# B&R Automation Studio project 8238
Automation Studio 4.10.2.37; technology packages: mapp 5.15.0, mappSafety 5.15.0, mappView 5.15.1, mappVision 5.15.0

## Configuration LargeLoop

CPU , AutomationRuntime E4.34, Build 4.1.2, Safety 0.0, Vc V4.33.0

### Task classes (Cpu.sw)
```
Cyclic#1 (cycle 5000 us):
  Lift_PosMo <- Robo_Drive_Control.Lift_PosMonitor.prg [disabled]
  ServerTask <- (binary)
  USB_Pmem <- (binary)
  zzClearMem <- (binary)
  can_dry1 <- (binary)
  zzSQLid <- (binary)
  Belt_Test <- (binary)
Cyclic#2 (cycle 10000 us, tolerance 10000 us):
  IO_INPUTS <- IO_INPUTS.prg
  S_COMM_IN <- S_COMM_IN.prg
  DBOUNCE <- DBOUNCE.prg
  INSERTS <- INSERTS.prg
  WEIGHT <- WEIGHT.prg
  BRING_OK <- BRING_OK.prg
  LIFTS <- LIFTS.prg
  CLOSERS <- CLOSERS.prg
  SWITCHES <- SWITCHES.prg
  OPENERS <- OPENERS.prg
  RAIL_SUB <- RAIL_SUB.prg
  ALARMS <- ALARMS.prg
  IO_OUTPUTS <- IO_OUTPUTS.prg
  S_COMM_OUT <- S_COMM_OUT.prg
  Lift_v8_1 <- Robo_Drive_Control.Lift_v8_1.prg
  custom <- custom.prg
  zzStd <- Standard.Standard.zzStd.prg
Cyclic#8 (cycle 5000 us):
  ModSlave <- ModSlave.prg
DataObjects: Param_1_5k <- Robo_Drive_Control.Param_1_5kwStar_expo.dob, assl1, arsdmsvp, arsdmhtm, arsdmsvg
Binaries: TCData, udbdef, ashwac, User, Role, OpcUaMap, asfw, arconfig, iomap, ashwd, sysconf, vcfntttf, vcfile, vcshared, vccshape, vcgclass, arial, CT1102, vcchspot, vcdsint, PCT0403, vccbtn, vcdsloc, vccovl, vccline, vcctext, vcalarm, vcbclass, vcrt, vccnum, vccstr, CT1103, arialbd, PCT0402, vcpdsw, verdanab, verdana, webserv, arsdm
Libraries: FC302, MbusTCP, sys_lib, AsARCfg, AsTCP, asstring, AsCANopen, runtime, standard, asieccon, astime, vcresman, WETCAN2, MTTypes, brsystem
```

### Hardware
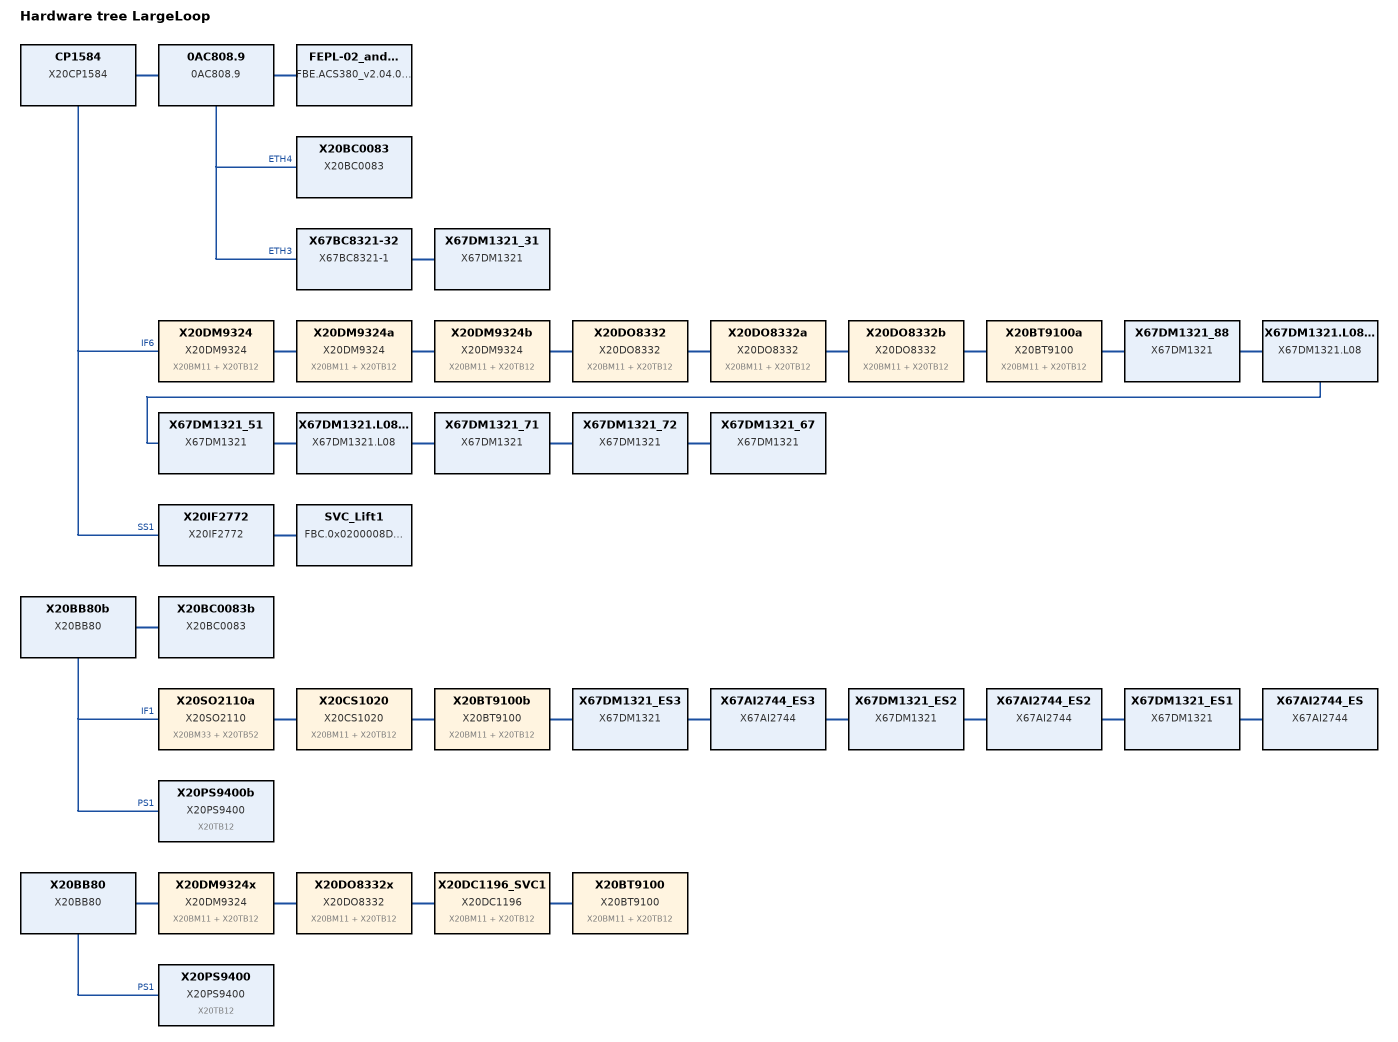
```
0AC808.9 : 0AC808.9 v1.0.0.0  [ETH1 -> CP1584.IF3 [Cable Type=PowerlinkCable, Length=10, Version=1.0.0.3]; ETH3 -> X67BC8321-32.PLK1 [Cable Type=PowerlinkCable, Length=10, Version=1.0.0.3]; ETH4 -> X20BC0083.PLK1 [Cable Type=PowerlinkCable, Length=10, Version=1.0.0.3]; ETH7 -> FEPL-02_and_ACS380_STB1.PLK1 [Cable Type=PowerlinkCable, Length=10, Version=1.0.0.3]]
CP1584 : X20CP1584 v1.9.0.0
  Connector IF2:
    ActivateDevice = 1
    Mode = Manual
    InternetAddress = 10.8.4.20
    SubnetMask = 
  Connector IF3:
    DNAConfiguration = manual
    InternetAddress = 10.0.20.20
    SubnetMask = 255.255.255.0
    ActivateIna = 1
    InaNodeNumber = 21
  Connector IF6:
    Stations = 100
  ConfigurationID = AS4_2_BaseStandard_Supertrack
  UserRamSize = 966656
  RemMemSize = 65280
  PermanentPvSize = 46956
  RemanentGlobalPvSize = 12000
  VolatileGlobalPvSize = 400000
  CyclicObjects = 200
  BRObjects = 600
  EnableUsbRemoteInstall = 1
  EnableCfRemoteInstall = 1
  Cyclic1Duration = 5000
  Cyclic2Duration = 10000
  Cyclic2Tolerance = 10000
  Cyclic8Duration = 5000
  FileDevice1
  FileDeviceName1 = USBStick
  FileDevicePath1 = /bd0\
  EthernetHostName = SupertrackPLC
  EthernetDefaultGateway = 10.8.15.254
  ActivateOpcUa = 1
  OpcUa_Security_SoftwareCertificates = 
  OpcUaInformationModels_PV_Version = 1
FEPL-02_and_ACS380_STB1 : FBE.ACS380_v2.04.0.3_FEPL-02_1.0_filerev1.0 vFFEPS10 (OrderNumber=FEPL-02 and ACS380)  [PLK1 -> 0AC808.9.ETH7 (NodeNumber=101) [Cable Type=PowerlinkCable, Length=10, Version=1.0.0.3]]
  Supervision = off
  p2201_direction = ro
  p2203_direction = ro
  p6040_direction = wo
  p6041_direction = ro
  p6042_direction = wo
  p6044_direction = ro
  p4001s07_direction = ro
  p4001s0A_direction = ro
  p401Cs48_direction = wo
  p401Cs49_direction = wo
  p4063s06_direction = wo
  p4063s09_direction = wo
  p4063s0A_direction = wo
SVC_Lift1 : FBC.0x0200008D.0x00000064.CO302A_4 v0x04.0x2A (OrderNumber=MCA105 CANopen)  [CAN1 -> X20IF2772.IF1 (NodeNumber=11)]
  p6040_connecttomaster = 6
  p6041_connecttomaster = 2
  p1400_transmissionselection = 0
  p1401_transmissionselection = 1
  p1402_transmissionselection = 0
  p1403_transmissionselection = 0
  p1800_transmissionselection = 0
  p1801_transmissionselection = 1
  p1802_transmissionselection = 0
  p1803_transmissionselection = 1
  pheartbeat_producertime = 500
  p241a_subnumber = 0x08
  p241a_parametername = 1050. Process Data Con
  p241a_objecttype = 8
  p241a_objflags = 0
  p241a_parametervalue = 
  p241asub0_parametername = 1050. Process Data Con index 0
  p241asub0_objecttype = 7
  p241asub0_accesstype = RW
  p241asub0_datatype = 6
  p241asub0_pdomapping = 0
  p241asub0_objflags = 0
  p241asub0_lowlimit = 0x0
  p241asub0_highlimit = 0x7d0
  p241asub0_parametervalue = 
  p241asub1_parametername = 1050. Process Data Con index 1
  p241asub1_objecttype = 7
  p241asub1_accesstype = RW
  p241asub1_datatype = 6
  p241asub1_pdomapping = 0
  p241asub1_objflags = 0
  p241asub1_lowlimit = 0x0
  p241asub1_highlimit = 0x7d0
  p241asub1_parametervalue = 
  p241asub2_parametername = 1050. Process Data Con index 2
  p241asub2_objecttype = 7
  p241asub2_accesstype = RW
  p241asub2_datatype = 6
  p241asub2_pdomapping = 0
  p241asub2_objflags = 0
  p241asub2_lowlimit = 0x0
  p241asub2_highlimit = 0x7d0
  p241asub2_parametervalue = 
  p241asub3_parametername = 1050. Process Data Con index 3
  p241asub3_objecttype = 7
  p241asub3_accesstype = RW
  p241asub3_datatype = 6
  p241asub3_pdomapping = 0
  p241asub3_objflags = 0
  p241asub3_lowlimit = 0x0
  p241asub3_highlimit = 0x7d0
  p241asub3_parametervalue = 
  p241asub4_parametername = 1050. Process Data Con index 4
  p241asub4_objecttype = 7
  p241asub4_accesstype = RW
  p241asub4_datatype = 6
  p241asub4_pdomapping = 0
  p241asub4_objflags = 0
  p241asub4_lowlimit = 0x0
  p241asub4_highlimit = 0x7d0
  p241asub4_parametervalue = 
  p241asub5_parametername = 1050. Process Data Con index 5
  p241asub5_objecttype = 7
  p241asub5_accesstype = RW
  p241asub5_datatype = 6
  p241asub5_pdomapping = 0
  p241asub5_objflags = 0
  p241asub5_lowlimit = 0x0
  p241asub5_highlimit = 0x7d0
  p241asub5_parametervalue = 
  p241asub6_parametername = 1050. Process Data Con index 6
  p241asub6_objecttype = 7
  p241asub6_accesstype = RW
  p241asub6_datatype = 6
  p241asub6_pdomapping = 0
  p241asub6_objflags = 0
  p241asub6_lowlimit = 0x0
  p241asub6_highlimit = 0x7d0
  p241asub6_parametervalue = 
  p241asub7_parametername = 1050. Process Data Con index 7
  p241asub7_objecttype = 7
  p241asub7_accesstype = RW
  p241asub7_datatype = 6
  p241asub7_pdomapping = 0
  p241asub7_objflags = 0
  p241asub7_lowlimit = 0x0
  p241asub7_highlimit = 0x7d0
  p241asub7_parametervalue = 
  p241b_subnumber = 0x08
  p241b_parametername = 1051. Process Data Con
  p241b_objecttype = 8
  p241b_objflags = 0
  p241b_parametervalue = 
  p241bsub0_parametername = 1051. Process Data Con index 0
  p241bsub0_objecttype = 7
  p241bsub0_accesstype = RW
  p241bsub0_datatype = 6
  p241bsub0_pdomapping = 0
  p241bsub0_objflags = 0
  p241bsub0_lowlimit = 0x0
  p241bsub0_highlimit = 0x7d0
  p241bsub0_parametervalue = 
  p241bsub1_parametername = 1051. Process Data Con index 1
  p241bsub1_objecttype = 7
  p241bsub1_accesstype = RW
  p241bsub1_datatype = 6
  p241bsub1_pdomapping = 0
  p241bsub1_objflags = 0
  p241bsub1_lowlimit = 0x0
  p241bsub1_highlimit = 0x7d0
  p241bsub1_parametervalue = 
  p241bsub2_parametername = 1051. Process Data Con index 2
  p241bsub2_objecttype = 7
  p241bsub2_accesstype = RW
  p241bsub2_datatype = 6
  p241bsub2_pdomapping = 0
  p241bsub2_objflags = 0
  p241bsub2_lowlimit = 0x0
  p241bsub2_highlimit = 0x7d0
  p241bsub2_parametervalue = 
  p241bsub3_parametername = 1051. Process Data Con index 3
  p241bsub3_objecttype = 7
  p241bsub3_accesstype = RW
  p241bsub3_datatype = 6
  p241bsub3_pdomapping = 0
  p241bsub3_objflags = 0
  p241bsub3_lowlimit = 0x0
  p241bsub3_highlimit = 0x7d0
  p241bsub3_parametervalue = 
  p241bsub4_parametername = 1051. Process Data Con index 4
  p241bsub4_objecttype = 7
  p241bsub4_accesstype = RW
  p241bsub4_datatype = 6
  p241bsub4_pdomapping = 0
  p241bsub4_objflags = 0
  p241bsub4_lowlimit = 0x0
  p241bsub4_highlimit = 0x7d0
  p241bsub4_parametervalue = 
  p241bsub5_parametername = 1051. Process Data Con index 5
  p241bsub5_objecttype = 7
  p241bsub5_accesstype = RW
  p241bsub5_datatype = 6
  p241bsub5_pdomapping = 0
  p241bsub5_objflags = 0
  p241bsub5_lowlimit = 0x0
  p241bsub5_highlimit = 0x7d0
  p241bsub5_parametervalue = 
  p241bsub6_parametername = 1051. Process Data Con index 6
  p241bsub6_objecttype = 7
  p241bsub6_accesstype = RW
  p241bsub6_datatype = 6
  p241bsub6_pdomapping = 0
  p241bsub6_objflags = 0
  p241bsub6_lowlimit = 0x0
  p241bsub6_highlimit = 0x7d0
  p241bsub6_parametervalue = 
  p241bsub7_parametername = 1051. Process Data Con index 7
  p241bsub7_objecttype = 7
  p241bsub7_accesstype = RW
  p241bsub7_datatype = 6
  p241bsub7_pdomapping = 0
  p241bsub7_objflags = 0
  p241bsub7_lowlimit = 0x0
  p241bsub7_highlimit = 0x7d0
  p241bsub7_parametervalue = 
X20BB80 : X20BB80 v1.1.0.0
X20BB80b : X20BB80 v1.1.0.0
X20BC0083 : X20BC0083 v2.14.0.0  [PLK1 -> 0AC808.9.ETH4 (NodeNumber=2) [Cable Type=PowerlinkCable, Length=10, Version=1.0.0.3]; SL -> X20BB80.SL1]
  Supervision = off
X20BC0083b : X20BC0083 v2.14.0.0  [SL -> X20BB80b.SL1]
  Supervision = off
X20BM11 : X20BM11 v1.0.0.1  [X2X1 -> CP1584.IF6]
X20BM11a : X20BM11 v1.0.0.1  [X2X1 -> X20BM11.X2X2]
X20BM11b : X20BM11 v1.0.0.1  [X2X1 -> X20BB80.IF1]
X20BM11c : X20BM11 v1.0.0.1  [X2X1 -> X20BM33b.X2X2]
X20BM11d : X20BM11 v1.0.0.1  [X2X1 -> X20BM11a.X2X2]
X20BM11e : X20BM11 v1.0.0.1  [X2X1 -> X20BM11d.X2X2]
X20BM11f : X20BM11 v1.0.0.1  [X2X1 -> X20BM11e.X2X2]
X20BM11g : X20BM11 v1.0.0.1  [X2X1 -> X20BM11b.X2X2]
X20BM11h : X20BM11 v1.0.0.1  [X2X1 -> X20BM11f.X2X2]
X20BM11i : X20BM11 v1.0.0.1  [X2X1 -> X20BM11g.X2X2]
X20BM11j : X20BM11 v1.0.0.1  [X2X1 -> X20BM11i.X2X2]
X20BM11k : X20BM11 v1.0.0.1  [X2X1 -> X20BM11h.X2X2]
X20BM11l : X20BM11 v1.0.0.1  [X2X1 -> X20BM11c.X2X2]
X20BM33b : X20BM33 v1.1.0.0  [X2X1 -> X20BB80b.IF1]
X20BT9100 : X20BT9100 v1.1.0.0  [SS1 -> X20TB12k.SS; SL -> X20BM11j.SL1]
  Supervision = off
X20BT9100a : X20BT9100 v1.1.0.0  [SS1 -> X20TB12l.SS; SL -> X20BM11k.SL1]
  Supervision = off
X20BT9100b : X20BT9100 v1.1.0.0  [SS1 -> X20TB12d.SS; SL -> X20BM11l.SL1]
  Supervision = off
X20CS1020 : X20CS1020 v1.7.0.0  [SS1 -> X20TB12o.SS; SL -> X20BM11c.SL1]
  Supervision = off
X20DC1196_SVC1 : X20DC1196 v1.3.0.0  [SS1 -> X20TB12j.SS; SL -> X20BM11i.SL1]
  FunctionModel = FunctionModel001
  Supervision = off
X20DM9324 : X20DM9324 v1.0.4.0  [SS1 -> X20TB12a.SS; SL -> X20BM11.SL1]
  Supervision = off
X20DM9324a : X20DM9324 v1.0.4.0  [SS1 -> X20TB12b.SS; SL -> X20BM11a.SL1]
  Supervision = off
X20DM9324b : X20DM9324 v1.0.4.0  [SS1 -> X20TB12e.SS; SL -> X20BM11d.SL1]
  Supervision = off
X20DM9324x : X20DM9324 v1.0.4.0  [SS1 -> X20TB12c.SS; SL -> X20BM11b.SL1]
  Supervision = off
X20DO8332 : X20DO8332 v1.0.2.0  [SS1 -> X20TB12f.SS; SL -> X20BM11e.SL1]
  Supervision = off
X20DO8332a : X20DO8332 v1.0.2.0  [SS1 -> X20TB12g.SS; SL -> X20BM11f.SL1]
  Supervision = off
X20DO8332b : X20DO8332 v1.0.2.0  [SS1 -> X20TB12i.SS; SL -> X20BM11h.SL1]
  Supervision = off
X20DO8332x : X20DO8332 v1.0.2.0  [SS1 -> X20TB12h.SS; SL -> X20BM11g.SL1]
  Supervision = off
X20IF2772 : X20IF2772 v1.5.0.0  [SS -> CP1584.SS1]
  Connector IF1:
    Baudrate = 250000
    ActivateCANIO = 0
    ActivateCanOpen = 1
    pcannodeid = 2
    pnmtstartup_bit3 = 1
    pnmtstartup_maximumbootuptime = 20
    pheartbeat_producertime = 500
    pactivatesync = 1
    pcycleperiod = 10000
    pwindowlength = 10000
    p1006_parametervalue = 0
    p1007_parametervalue = 0
    p100c_parametervalue = 1000
    p100d_parametervalue = 3
  Connector IF2:
    Baudrate = 250000
    ActivateCanOpen = 1
    pcannodeid = 3
    p1006_parametervalue = 0
    p1007_parametervalue = 0
    p100c_parametervalue = 1000
    p100d_parametervalue = 3
X20PS9400 : X20PS9400 v1.7.0.0  [SS1 -> X20TB12.SS; PS -> X20BB80.PS1]
  Supervision = off
X20PS9400b : X20PS9400 v1.7.0.0  [SS1 -> X20TB12m.SS; PS -> X20BB80b.PS1]
  Supervision = off
X20SO2110a : X20SO2110 v2.2.1.0  [SS1 -> X20TB52d.SS; SL -> X20BM33b.SL1]
  Supervision = off
  SafeModuleID = 4
X20TB12 : X20TB12 v1.0.0.0
X20TB12a : X20TB12 v1.0.0.0
X20TB12b : X20TB12 v1.0.0.0
X20TB12c : X20TB12 v1.0.0.0
X20TB12d : X20TB12 v1.0.0.0
X20TB12e : X20TB12 v1.0.0.0
X20TB12f : X20TB12 v1.0.0.0
X20TB12g : X20TB12 v1.0.0.0
X20TB12h : X20TB12 v1.0.0.0
X20TB12i : X20TB12 v1.0.0.0
X20TB12j : X20TB12 v1.0.0.0
X20TB12k : X20TB12 v1.0.0.0
X20TB12l : X20TB12 v1.0.0.0
X20TB12m : X20TB12 v1.0.0.0
X20TB12o : X20TB12 v1.0.0.0
X20TB52d : X20TB52 v1.0.0.2
X67AI2744_ES : X67AI2744 v1.3.0.0  [X2X1 -> X67DM1321_ES1.X2X2 [Cable Type=X2XCable, Length=10, Version=1.0.0.3]]
  Supervision = off
X67AI2744_ES2 : X67AI2744 v1.3.0.0  [X2X1 -> X67DM1321_ES2.X2X2 [Cable Type=X2XCable, Length=10, Version=1.0.0.3]]
  Supervision = off
X67AI2744_ES3 : X67AI2744 v1.3.0.0  [X2X1 -> X67DM1321_ES3.X2X2 [Cable Type=X2XCable, Length=10, Version=1.0.0.3]]
  Supervision = off
X67BC8321-32 : X67BC8321-1 v2.14.0.0  [PLK1 -> 0AC808.9.ETH3 (NodeNumber=1) [Cable Type=PowerlinkCable, Length=10, Version=1.0.0.3]]
  IOSupervision = off
  Direction05 = output
  Direction07 = output
  Direction08 = output
X67DM1321.L08_151 : X67DM1321.L08 v1.3.0.0  [X2X1 -> X67DM1321_88.X2X2 [Cable Type=X2XCable, Length=10, Version=1.0.0.3]]
  Supervision = off
  Direction09 = output
  Direction10 = output
  Direction11 = output
  Direction12 = output
  Direction13 = output
  Direction14 = output
  Direction15 = output
  Direction16 = output
X67DM1321.L08_152 : X67DM1321.L08 v1.3.0.0  [X2X1 -> X67DM1321_51.X2X2 [Cable Type=X2XCable, Length=10, Version=1.0.0.3]]
  Supervision = off
  Direction09 = output
  Direction10 = output
  Direction11 = output
  Direction12 = output
  Direction13 = output
  Direction14 = output
  Direction15 = output
  Direction16 = output
X67DM1321_31 : X67DM1321 v1.2.0.0  [X2X1 -> X67BC8321-32.IF1 [Cable Type=X2XCable, Length=10, Version=1.0.0.3]]
  Supervision = off
  Direction08 = output
X67DM1321_51 : X67DM1321 v1.2.0.0  [X2X1 -> X67DM1321.L08_151.X2X2 [Cable Type=X2XCable, Length=10, Version=1.0.0.3]]
  Supervision = off
  Direction05 = output
  Direction06 = output
  Direction07 = output
  Direction08 = output
X67DM1321_67 : X67DM1321 v1.2.0.0  [X2X1 -> X67DM1321_72.X2X2 [Cable Type=X2XCable, Length=10, Version=1.0.0.3]]
  Supervision = off
  Direction04 = output
  Direction05 = output
  Direction06 = output
  Direction07 = output
  Direction08 = output
X67DM1321_71 : X67DM1321 v1.2.0.0  [X2X1 -> X67DM1321.L08_152.X2X2 [Cable Type=X2XCable, Length=10, Version=1.0.0.3]]
  Supervision = off
  Direction03 = output
  Direction04 = output
  Direction05 = output
  Direction06 = output
  Direction07 = output
  Direction08 = output
X67DM1321_72 : X67DM1321 v1.2.0.0  [X2X1 -> X67DM1321_71.X2X2 [Cable Type=X2XCable, Length=10, Version=1.0.0.3]]
  Supervision = off
  Direction03 = output
  Direction04 = output
  Direction05 = output
  Direction06 = output
  Direction07 = output
  Direction08 = output
X67DM1321_88 : X67DM1321 v1.2.0.0  [X2X1 -> X20BT9100a.X2X1 [Cable Type=X2XCable, Length=10, Version=1.0.0.3]]
  Supervision = off
  Direction06 = output
  Direction07 = output
  Direction08 = output
X67DM1321_ES1 : X67DM1321 v1.2.0.0  [X2X1 -> X67AI2744_ES2.X2X2 [Cable Type=X2XCable, Length=10, Version=1.0.0.3]]
  Supervision = off
  Direction01 = output
  Direction02 = output
  Direction05 = output
  Direction06 = output
  Direction07 = output
  Direction08 = output
X67DM1321_ES2 : X67DM1321 v1.2.0.0  [X2X1 -> X67AI2744_ES3.X2X2 [Cable Type=X2XCable, Length=10, Version=1.0.0.3]]
  Supervision = off
  Direction01 = output
  Direction02 = output
  Direction05 = output
  Direction06 = output
  Direction07 = output
  Direction08 = output
X67DM1321_ES3 : X67DM1321 v1.2.0.0  [X2X1 -> X20BT9100b.X2X1 [Cable Type=X2XCable, Length=10, Version=1.0.0.3]]
  Supervision = off
  Direction01 = output
  Direction02 = output
  Direction05 = output
  Direction06 = output
  Direction07 = output
  Direction08 = output
```

### IoMap.iom - CP1584/IoMap.iom
```iecst
(********************************************************************
 * COPYRIGHT --
 ********************************************************************
 * File: IoMap.iom
 * Author: Dave
 * Created: November 19, 2010
 ********************************************************************
 * IO mapping file
 ********************************************************************)
VAR_CONFIG
	OK[1] AT %IX."X20DM9324x".ModuleOk;
	OK[3] AT %IX."X20DO8332x".ModuleOk;
	X[1].X01 AT %IX."X20DM9324x".DigitalInput01; (*Emergency stops Ok*)
	X[1].X02 AT %IX."X20DM9324x".DigitalInput02; (*Motor overloads*)
	X[1].X03 AT %IX."X20DM9324x".DigitalInput03; (*SR1 Ok*)
	X[1].X04 AT %IX."X20DM9324x".DigitalInput04; (*Spare*)
	X[1].X05 AT %IX."X20DM9324x".DigitalInput05; (*STB1 - PX*)
	X[1].X06 AT %IX."X20DM9324x".DigitalInput06; (*STB2 -PX*)
	X[1].X07 AT %IX."X20DM9324x".DigitalInput07; (*ES2 - Emergency stop*)
	X[1].X08 AT %IX."X20DM9324x".DigitalInput08; (*ES3 - Emergency stop*)
	Y[1].Y01 AT %QX."X20DM9324x".DigitalOutput01; (*Alarm beacon*)
	Y[1].Y02 AT %QX."X20DM9324x".DigitalOutput02; (*Spare*)
	Y[1].Y03 AT %QX."X20DM9324x".DigitalOutput03; (*Spare*)
	Y[1].Y04 AT %QX."X20DM9324x".DigitalOutput04; (*Spare*)
	Y[3].Y01 AT %QX."X20DO8332x".DigitalOutput01; (*STB1 - Run*)
	Y[3].Y02 AT %QX."X20DO8332x".DigitalOutput02; (*STB2 - Run*)
	Y[3].Y03 AT %QX."X20DO8332x".DigitalOutput03; (*Spare*)
	Y[3].Y04 AT %QX."X20DO8332x".DigitalOutput04; (*Spare*)
	Y[3].Y05 AT %QX."X20DO8332x".DigitalOutput05; (*Spare*)
	Y[3].Y06 AT %QX."X20DO8332x".DigitalOutput06; (*SVC1 - Carriage stop*)
	Y[3].Y07 AT %QX."X20DO8332x".DigitalOutput07; (*Spare*)
	Y[3].Y08 AT %QX."X20DO8332x".DigitalOutput08; (*Spare*)
	X[32].X01 AT %IX."X67BC8321-32".IF1.ST1.DigitalInput01; (*SVC1 - Over travel top*)
	X[32].X02 AT %IX."X67BC8321-32".IF1.ST1.DigitalInput02; (*Spare*)
	X[32].X03 AT %IX."X67BC8321-32".IF1.ST1.DigitalInput03; (*SVC1 - Over travel bottom*)
	Cyclic#1.X[32].X04 AT %IX."X67BC8321-32".IF1.ST1.DigitalInput04; (*SVC1 - Reference switch*)
	Y[32].Y05 AT %QX."X67BC8321-32".IF1.ST1.DigitalOutput05; (*SVC1 - Rail end stop (Empty bag in)*)
	Y[32].Y07 AT %QX."X67BC8321-32".IF1.ST1.DigitalOutput07; (*Spare*)
	Y[32].Y08 AT %QX."X67BC8321-32".IF1.ST1.DigitalOutput08; (*SVC1 - Open buffer stop*)
	OK[31] AT %IX."X67DM1321_31".ModuleOk;
	X[31].X01 AT %IX."X67DM1321_31".DigitalInput01; (*Spare*)
	X[31].X02 AT %IX."X67DM1321_31".DigitalInput02; (*Spare*)
	X[31].X03 AT %IX."X67DM1321_31".DigitalInput03; (*Spare*)
	X[31].X04 AT %IX."X67DM1321_31".DigitalInput04; (*SVC1 Bag arrive on carriage*)
	X[31].X05 AT %IX."X67DM1321_31".DigitalInput05; (*SVC1 Bag on carriage*)
	X[31].X06 AT %IX."X67DM1321_31".DigitalInput06; (*SVC1 Rail align receive*)
	X[31].X07 AT %IX."X67DM1321_31".DigitalInput07; (*SVC1 Rail align release*)
	Y[31].Y08 AT %QX."X67DM1321_31".DigitalOutput08; (*Spare*)
	X[32].X06 AT %IX."X67BC8321-32".IF1.ST1.DigitalInput06; (*SVC1 - Bag at buffer*)
	X[88].X01 AT %IX."X67DM1321_88".DigitalInput01; (*Spare*)
	X[88].X02 AT %IX."X67DM1321_88".DigitalInput02; (*STRF1 - Bag at buffer*)
	X[88].X03 AT %IX."X67DM1321_88".DigitalInput03; (*STRF1 - Bag arrive*)
	X[88].X04 AT %IX."X67DM1321_88".DigitalInput04; (*STRF1 - Bag past point*)
	Y[88].Y06 AT %QX."X67DM1321_88".DigitalOutput06; (*STRF1 - Open buffer*)
	Y[88].Y07 AT %QX."X67DM1321_88".DigitalOutput07; (*STRF1 - Select line B*)
	Y[88].Y08 AT %QX."X67DM1321_88".DigitalOutput08; (*STRF1 - Select line A*)
	OK[88] AT %IX."X67DM1321_88".ModuleOk;
	X[151].X01 AT %IX."X67DM1321.L08_151".DigitalInput01; (*SDC1 - Bag at buffer*)
	X[151].X02 AT %IX."X67DM1321.L08_151".DigitalInput02; (*SDC1 - Bag at Discharger*)
	X[151].X03 AT %IX."X67DM1321.L08_151".DigitalInput03; (*SDC1 - Bag released*)
	X[151].X04 AT %IX."X67DM1321.L08_151".DigitalInput04; (*SDC1 - Bag empty*)
	X[151].X05 AT %IX."X67DM1321.L08_151".DigitalInput05; (*Spare*)
	X[151].X06 AT %IX."X67DM1321.L08_151".DigitalInput06; (*SDC1 - Drop load pushbutton*)
	X[151].X07 AT %IX."X67DM1321.L08_151".DigitalInput07; (*Spare*)
	X[151].X08 AT %IX."X67DM1321.L08_151".DigitalInput08; (*Spare*)
	Y[151].Y01 AT %QX."X67DM1321.L08_151".DigitalOutput09; (*SDC1 - Open buffer stop*)
	Y[151].Y02 AT %QX."X67DM1321.L08_151".DigitalOutput10; (*SDC1 - Bag steady*)
	Y[151].Y03 AT %QX."X67DM1321.L08_151".DigitalOutput11; (*SDC1 - Open bag*)
	Y[151].Y04 AT %QX."X67DM1321.L08_151".DigitalOutput12; (*SDC1 - Open stop*)
	Y[151].Y05 AT %QX."X67DM1321.L08_151".DigitalOutput13; (*SDC1 - Bag closer*)
	Y[151].Y06 AT %QX."X67DM1321.L08_151".DigitalOutput14; (*SSB1 Bag catch*)
	Y[151].Y07 AT %QX."X67DM1321.L08_151".DigitalOutput15; (*SSB1 Close bag*)
	Y[151].Y08 AT %QX."X67DM1321.L08_151".DigitalOutput16; (*SDC1 - Pushbutton lamp*)
	OK[151] AT %IX."X67DM1321.L08_151".ModuleOk;
	X[88].X05 AT %IX."X67DM1321_88".DigitalInput05; (*STRF1 - Bag released*)
	X[51].X01 AT %IX."X67DM1321_51".DigitalInput01; (*SPN1 - Bag arrive line 1*)
	X[51].X02 AT %IX."X67DM1321_51".DigitalInput02; (*SPN1 - Bag arrive line 2*)
	X[51].X03 AT %IX."X67DM1321_51".DigitalInput03; (*SPN1 - Bag arrive line 3*)
	X[51].X04 AT %IX."X67DM1321_51".DigitalInput04; (*Spare*)
	Y[51].Y05 AT %QX."X67DM1321_51".DigitalOutput05; (*SPN1 - Select line 3*)
	Y[51].Y06 AT %QX."X67DM1321_51".DigitalOutput06; (*SPN1 - Select line 2*)
	Y[51].Y07 AT %QX."X67DM1321_51".DigitalOutput07; (*SPN1 - Reset line 3*)
	Y[51].Y08 AT %QX."X67DM1321_51".DigitalOutput08; (*SPN1 - Reset line 2*)
	OK[51] AT %IX."X67DM1321_51".ModuleOk;
	X[152].X01 AT %IX."X67DM1321.L08_152".DigitalInput01; (*SDC2 - Bag at buffer*)
	X[152].X02 AT %IX."X67DM1321.L08_152".DigitalInput02; (*SDC2 - Bag at Discharger*)
	X[152].X03 AT %IX."X67DM1321.L08_152".DigitalInput03; (*SDC2 - Bag released*)
	X[152].X04 AT %IX."X67DM1321.L08_152".DigitalInput04; (*SDC2 - Bag empty*)
	X[152].X05 AT %IX."X67DM1321.L08_152".DigitalInput05; (*Spare*)
	X[152].X06 AT %IX."X67DM1321.L08_152".DigitalInput06; (*SDC2 - Drop load pushbutton*)
	X[152].X07 AT %IX."X67DM1321.L08_152".DigitalInput07; (*Spare*)
	X[152].X08 AT %IX."X67DM1321.L08_152".DigitalInput08; (*Spare*)
	Y[152].Y01 AT %QX."X67DM1321.L08_152".DigitalOutput09; (*SDC2 - Open buffer stop*)
	Y[152].Y02 AT %QX."X67DM1321.L08_152".DigitalOutput10; (*SDC2 - Bag steady*)
	Y[152].Y03 AT %QX."X67DM1321.L08_152".DigitalOutput11; (*SDC2 - Open bag*)
	Y[152].Y04 AT %QX."X67DM1321.L08_152".DigitalOutput12; (*SDC2 - Open stop*)
	Y[152].Y05 AT %QX."X67DM1321.L08_152".DigitalOutput13; (*SDC2 - Bag closer*)
	Y[152].Y06 AT %QX."X67DM1321.L08_152".DigitalOutput14; (*SSB2 Bag catch*)
	Y[152].Y07 AT %QX."X67DM1321.L08_152".DigitalOutput15; (*SSB2 Close bag*)
	Y[152].Y08 AT %QX."X67DM1321.L08_152".DigitalOutput16; (*SDC2 - Pushbutton lamp*)
	OK[152] AT %IX."X67DM1321.L08_152".ModuleOk;
	X[71].X01 AT %IX."X67DM1321_71".DigitalInput01; (*SPF1 - Bag at line 1*)
	X[71].X02 AT %IX."X67DM1321_71".DigitalInput02; (*SPF1 - Bag at line 2*)
	Y[71].Y03 AT %QX."X67DM1321_71".DigitalOutput03; (*SPF1 - Open stop  line 1*)
	Y[71].Y04 AT %QX."X67DM1321_71".DigitalOutput04; (*SPF1 - Open stop  line 2*)
	Y[71].Y05 AT %QX."X67DM1321_71".DigitalOutput05; (*Spare*)
	Y[71].Y06 AT %QX."X67DM1321_71".DigitalOutput06; (*SPF1 - Select line 2*)
	Y[71].Y07 AT %QX."X67DM1321_71".DigitalOutput07; (*Spare*)
	Y[71].Y08 AT %QX."X67DM1321_71".DigitalOutput08; (*SPF1 - Reset line 2*)
	OK[71] AT %IX."X67DM1321_71".ModuleOk; (*Module status (3 = module present)*)
	X[72].X01 AT %IX."X67DM1321_72".DigitalInput01; (*SPF1 - Bag at line 3*)
	X[72].X02 AT %IX."X67DM1321_72".DigitalInput02; (*SPF1 - Bag released*)
	Y[72].Y03 AT %QX."X67DM1321_72".DigitalOutput03; (*SPF1 - Open stop  line 3*)
	Y[72].Y04 AT %QX."X67DM1321_72".DigitalOutput04; (*Spare*)
	Y[72].Y05 AT %QX."X67DM1321_72".DigitalOutput05; (*SPF1 - Select line 3*)
	Y[72].Y06 AT %QX."X67DM1321_72".DigitalOutput06; (*Spare*)
	Y[72].Y07 AT %QX."X67DM1321_72".DigitalOutput07; (*SPF1 - Reset line 3*)
	Y[72].Y08 AT %QX."X67DM1321_72".DigitalOutput08; (*Spare*)
	OK[72] AT %IX."X67DM1321_72".ModuleOk; (*Module status (3 = module present)*)
	X[67].X01 AT %IX."X67DM1321_67".DigitalInput01; (*SVC2 - Bag at buffer line B*)
	X[67].X02 AT %IX."X67DM1321_67".DigitalInput02; (*SVC2 - Bag at buffer line A*)
	X[67].X03 AT %IX."X67DM1321_67".DigitalInput03; (*STRN1 - Bag past point*)
	Y[67].Y05 AT %QX."X67DM1321_67".DigitalOutput05; (*SVC2 - Open buffer line B*)
	Y[67].Y06 AT %QX."X67DM1321_67".DigitalOutput06; (*SVC2 - Open buffer line A*)
	Y[67].Y07 AT %QX."X67DM1321_67".DigitalOutput07; (*STRN1 - Select line B*)
	Y[67].Y08 AT %QX."X67DM1321_67".DigitalOutput08; (*STRN1 - Select line A*)
	OK[67] AT %IX."X67DM1321_67".ModuleOk;
	Y[67].Y04 AT %QX."X67DM1321_67".DigitalOutput04; (*SVC2 - Safety stops*)
	X[303].X03 AT %IX."X67DM1321_ES3".DigitalInput03; (*ES3 - Pushbutton*)
	X[303].X04 AT %IX."X67DM1321_ES3".DigitalInput04; (*Spare*)
	Y[303].Y01 AT %QX."X67DM1321_ES3".DigitalOutput01; (*ES3 - Lamp*)
	Y[303].Y02 AT %QX."X67DM1321_ES3".DigitalOutput02; (*ES3 - Open door*)
	Y[303].Y05 AT %QX."X67DM1321_ES3".DigitalOutput05; (*Spare*)
	Y[303].Y06 AT %QX."X67DM1321_ES3".DigitalOutput06; (*Spare*)
	Y[303].Y07 AT %QX."X67DM1321_ES3".DigitalOutput07; (*Spare*)
	Y[303].Y08 AT %QX."X67DM1321_ES3".DigitalOutput08; (*Spare*)
	OK[303] AT %IX."X67DM1321_ES3".ModuleOk;
	X[302].X03 AT %IX."X67DM1321_ES2".DigitalInput03; (*ES2 - Pushbutton*)
	X[302].X04 AT %IX."X67DM1321_ES2".DigitalInput04; (*Spare*)
	Y[302].Y01 AT %QX."X67DM1321_ES2".DigitalOutput01; (*ES2 - Lamp*)
	Y[302].Y02 AT %QX."X67DM1321_ES2".DigitalOutput02; (*ES2 - Open door*)
	Y[302].Y05 AT %QX."X67DM1321_ES2".DigitalOutput05; (*Spare*)
	Y[302].Y06 AT %QX."X67DM1321_ES2".DigitalOutput06; (*Spare*)
	Y[302].Y07 AT %QX."X67DM1321_ES2".DigitalOutput07; (*Spare*)
	Y[302].Y08 AT %QX."X67DM1321_ES2".DigitalOutput08; (*Spare*)
	OK[302] AT %IX."X67DM1321_ES2".ModuleOk;
	X[301].X03 AT %IX."X67DM1321_ES1".DigitalInput03; (*ES1 - Pushbutton*)
	X[301].X04 AT %IX."X67DM1321_ES1".DigitalInput04; (*Spare*)
	Y[301].Y01 AT %QX."X67DM1321_ES1".DigitalOutput01; (*ES1 - Lamp*)
	Y[301].Y02 AT %QX."X67DM1321_ES1".DigitalOutput02; (*ES1 - Open door*)
	Y[301].Y05 AT %QX."X67DM1321_ES1".DigitalOutput05; (*Spare*)
	Y[301].Y06 AT %QX."X67DM1321_ES1".DigitalOutput06; (*Spare*)
	Y[301].Y07 AT %QX."X67DM1321_ES1".DigitalOutput07; (*Spare*)
	Y[301].Y08 AT %QX."X67DM1321_ES1".DigitalOutput08; (*Spare*)
	OK[301] AT %IX."X67DM1321_ES1".ModuleOk;
	RB[1].Lift.CAN.ModuleOk AT %IX."SVC_Lift1".ModuleOk;
	RB[1].Lift.CAN.NodeStatus AT %IW."SVC_Lift1".NodeStatus;
	RB[1].Lift.CAN.ControlWord AT %QW."SVC_Lift1".CTW_6040_Out;
	RB[1].Lift.CAN.StatusWord AT %IW."SVC_Lift1".STW_6041;
	RB[1].Lift.CAN.TargetVelocity AT %QW."SVC_Lift1".TargetVelocity_6042_Out;
	RB[1].Lift.CAN.ControlEffort AT %IW."SVC_Lift1".ControlEffort_MAV_6044;
	RB[1].Lift.ModuleOK AT %IX."X20DC1196_SVC1".ModuleOk;
	RB[1].Lift.Encoder AT %ID."X20DC1196_SVC1".Encoder01;
  Cyclic#1.ABB_EPL[1].Comm.ModuleOk AT %IX."FEPL-02_and_ACS380_STB1".ModuleOk;
	Cyclic#1.ABB_EPL[1].Parameters.Write.Motor_NominalCurrent_9906 AT %QD."FEPL-02_and_ACS380_STB1"._9906_Motor_nominal_current_I4063_S06Out;
	Cyclic#1.ABB_EPL[1].Parameters.Write.Motor_NominalPower_9910 AT %QD."FEPL-02_and_ACS380_STB1"._9910_Motor_nominal_power_I4063_S0AOut;
	Cyclic#1.ABB_EPL[1].Parameters.Write.Motor_NominalSpeed_9909 AT %QD."FEPL-02_and_ACS380_STB1"._9909_Motor_nominal_speed_I4063_S09Out;
	Cyclic#1.ABB_EPL[1].Comm.ControlWord AT %QW."FEPL-02_and_ACS380_STB1".ControlWord_I6040Out;
	Cyclic#1.ABB_EPL[1].Comm.StatusWord AT %IW."FEPL-02_and_ACS380_STB1".StatusWord_I6041;
	Cyclic#1.ABB_EPL[1].Comm.ActVelocity AT %IW."FEPL-02_and_ACS380_STB1".VlVelocityActualValue_I6044;
	Cyclic#1.ABB_EPL[1].Comm.ActCurrent AT %ID."FEPL-02_and_ACS380_STB1"._0107_Motor_current_I4001_S07;
	Cyclic#1.ABB_EPL[1].Comm.ActTorque AT %ID."FEPL-02_and_ACS380_STB1"._0110_Motor_torque_I4001_S0A;
	Cyclic#1.ABB_EPL[1].Comm.ErrorCode AT %IW."FEPL-02_and_ACS380_STB1".VendorSpecificAlarmCodes_I2203;
	Cyclic#1.ABB_EPL[1].Parameters.Write.Ramp_AccTime1_2872 AT %QD."FEPL-02_and_ACS380_STB1"._2872_Freq_acceleration_time_1_I401C_S48Out;
	Cyclic#1.ABB_EPL[1].Parameters.Write.Ramp_DecTime1_2873 AT %QD."FEPL-02_and_ACS380_STB1"._2873_Freq_deceleration_time_1_I401C_S49Out;
	Cyclic#1.ABB_EPL[1].Comm.TargetVelocity AT %QW."FEPL-02_and_ACS380_STB1".VlTargetVelocity_I6042Out;
END_VAR
```

- Safety project (password-protected, skipped)

## Configuration eVue

CPU 5APC2200.AL14-000, AutomationRuntime D4.91, Build 4.1.2, Safety 0.0, Vc V4.62.0

### Task classes (Cpu.sw)
```
Cyclic#1 (cycle 1000 us, tolerance 2000 us):
  moduleWatc <- Standard.ModuleLogger.moduleWatch.prg
  USB_Pmem <- (binary)
  zzClearMem <- (binary)
  can_dry1 <- (binary)
  zzSQLid <- (binary)
  IO_Info <- (binary)
  IOLink_Dri <- (binary)
  SCANNERS <- (binary)
  SafetyUI <- (binary)
Cyclic#2 (cycle 12000 us, tolerance 12000 us):
  S_COMM_IN <- S_COMM_IN.prg
  IO_INPUTS <- IO_INPUTS.prg
  DBOUNCE <- DBOUNCE.prg
  custom <- custom.prg
  BELT_TO_TR <- BELT_TO_TRANSFER.prg
  CONVEYOR_M <- CONVEYOR_MAP.prg
  SAFETY_ZON <- SAFETY_ZONES.prg
  RAIL_SUB <- RAIL_SUB.prg
  LOADCELLS <- LOADCELLS.prg
  INSERTS <- INSERTS.prg
  WEIGHT <- WEIGHT.prg
  CLOSERS <- CLOSERS.prg
  OPENERS <- OPENERS.prg
  SWITCHES <- SWITCHES.prg
  LIFTS <- LIFTS.prg
  BRING_OK <- BRING_OK.prg
  Permenant <- Standard.Settings.Permenant.prg
  Lift_v8_1 <- Robo_Drive_Control.Lift_v8_1.prg [disabled]
  zzStd1 <- Standard.Standard.zzStd.prg
  FuseManage <- Standard.IOLink.Fuses.FuseManagement.prg
  Camera_Dri <- Standard.Barcode_BnR.Camera_Driver.prg [disabled]
  HoistServe <- Standard.HoistLibrary.HoistServer.prg
  hlKanLink <- Standard.Kanlink.KGFramework.Pkg_hlKanLink.hlKanLink.prg
Cyclic#4 (cycle 12000 us, tolerance 12000 us):
  WARNINGS <- WARNINGS.prg
Cyclic#5 (cycle 12000 us, tolerance 12000 us):
  ALARMS <- ALARMS.prg
Cyclic#6 (cycle 54000 us, tolerance 54000 us):
  zz_Kanlink <- Standard.Kanlink.zz_KanlinkConfig.prg
  Kan_Driver <- Standard.Kanlink.Kan_Driver.prg
  mnEth <- Standard.Kanlink.KGFramework.Pkg_mnEth.mnEth.prg
  svCPCache <- Standard.Kanlink.KGFramework.Pkg_svCPCache.svCPCache.prg
  kanlink_ma <- Standard.Kanlink.kanlink_map.prg
Cyclic#7 (cycle 102000 us, tolerance 102000 us):
  Contactron <- Standard.IOLink.Contactron.Contactron.prg
  httpServer <- http_Lib.httpServer.prg
Cyclic#8 (cycle 12000 us, tolerance 30000000 us):
  IO_OUTPUTS <- IO_OUTPUTS.prg
  S_COMM_OUT <- S_COMM_OUT.prg
  ModSlave <- COMMUNICATION.ModSlave.prg
  udpComm <- COMMUNICATION.UdpComm.prg
  tcpComm <- COMMUNICATION.TcpComm.prg
  udpComm_di <- SortingSpecial.udpComm_disp.prg
  zzGetTime <- CSP_Control.zzGetTime.prg
  OPCuAClien <- OPCuA_Client.OPCuAClient.prg
  mappSafety <- Safety.mappSafety.prg
  AccessCont <- Safety.AccessControl.prg
  Safety <- Safety.Safety.prg
  ABB_Driver <- Standard.ABB_EPL.ABB_Driver.prg
DataObjects: Param_1_5k <- Robo_Drive_Control.Param_1_5kwStar.dob [disabled], assl1, arsdmsvp, arsdmhtm, arsdmsvg
Binaries: mvLoader, TCLang, arflatprv, arcoal, TCData, udbdef, arsvcreg, FWRules, OpcUaSrv, Config, TC, viComp, Settings, viAppBCDE, cUnits, User, Role, sysconf, ashwd, arconfig, asfw, ashwac, iomap, Settings_1, Config_1, asiol1, asiol3, asiol2, asiol20, asiol17, asiol4, asiol19, asiol24, asiol30, asiol9, asiol12, asiol5, asiol29, asiol18, asiol16, asiol22, asiol6, asiol11, asiol28, asiol8, asiol26, asiol7, asiol15, asiol21, asiol10, asiol13, asiol32, asiol25, asiol31, asiol14, asiol23, asiol27, OpcUaMap, vcfntttf, vcfile, vcshared, vccshape, vcgclass, arial, CT1102, vcchspot, vcdsint, PCT0403, vccbtn, vcdsloc, vccovl, vccline, vcctext, vcalarm, vcbclass, vcrt, vccnum, vccstr, CT1103, arialbd, PCT0402, vcpdsw, verdanab, verdana, webserv, arsdm
Libraries: AsOpcUac, OPCuAClnt, FC302, standard, runtime, OPERATOR, AsTime, AsString, sys_lib, AsTCP, AsARCfg, AsIecCon, AsBrStr, FileIO, AsBrMath, CAN_Lib, AsUDP, MTTypes, brsystem, MpAudit, MpBase, DataObj, AsXml, MTBasics, MpServer, ArSsl, ArUser, ViBase, AsZip, powerlnk, AsEPL, AsETH, AsIODiag, AsHttp, AsIOAcc, AsIoTrc, FileMgr, AsIOLink, AsCANopen, AsIO, MbusTCP, SfDomain, KGstdLib, KGlibMsg, mnParamLib, KanLinkLib, KL_UserLib, libTestUse, AsBrWStr, ETHERNET, AsArLog, AsUSB, AsMem, AsDb, KanHttp, AsFifo, eVueLib, SfDomDrv, MpSfDomMgr, SfDomVis, SupFile, vcresman, WETCAN2, AsIOMMan, IOLinkLib, ABB_EPL
```

### Hardware
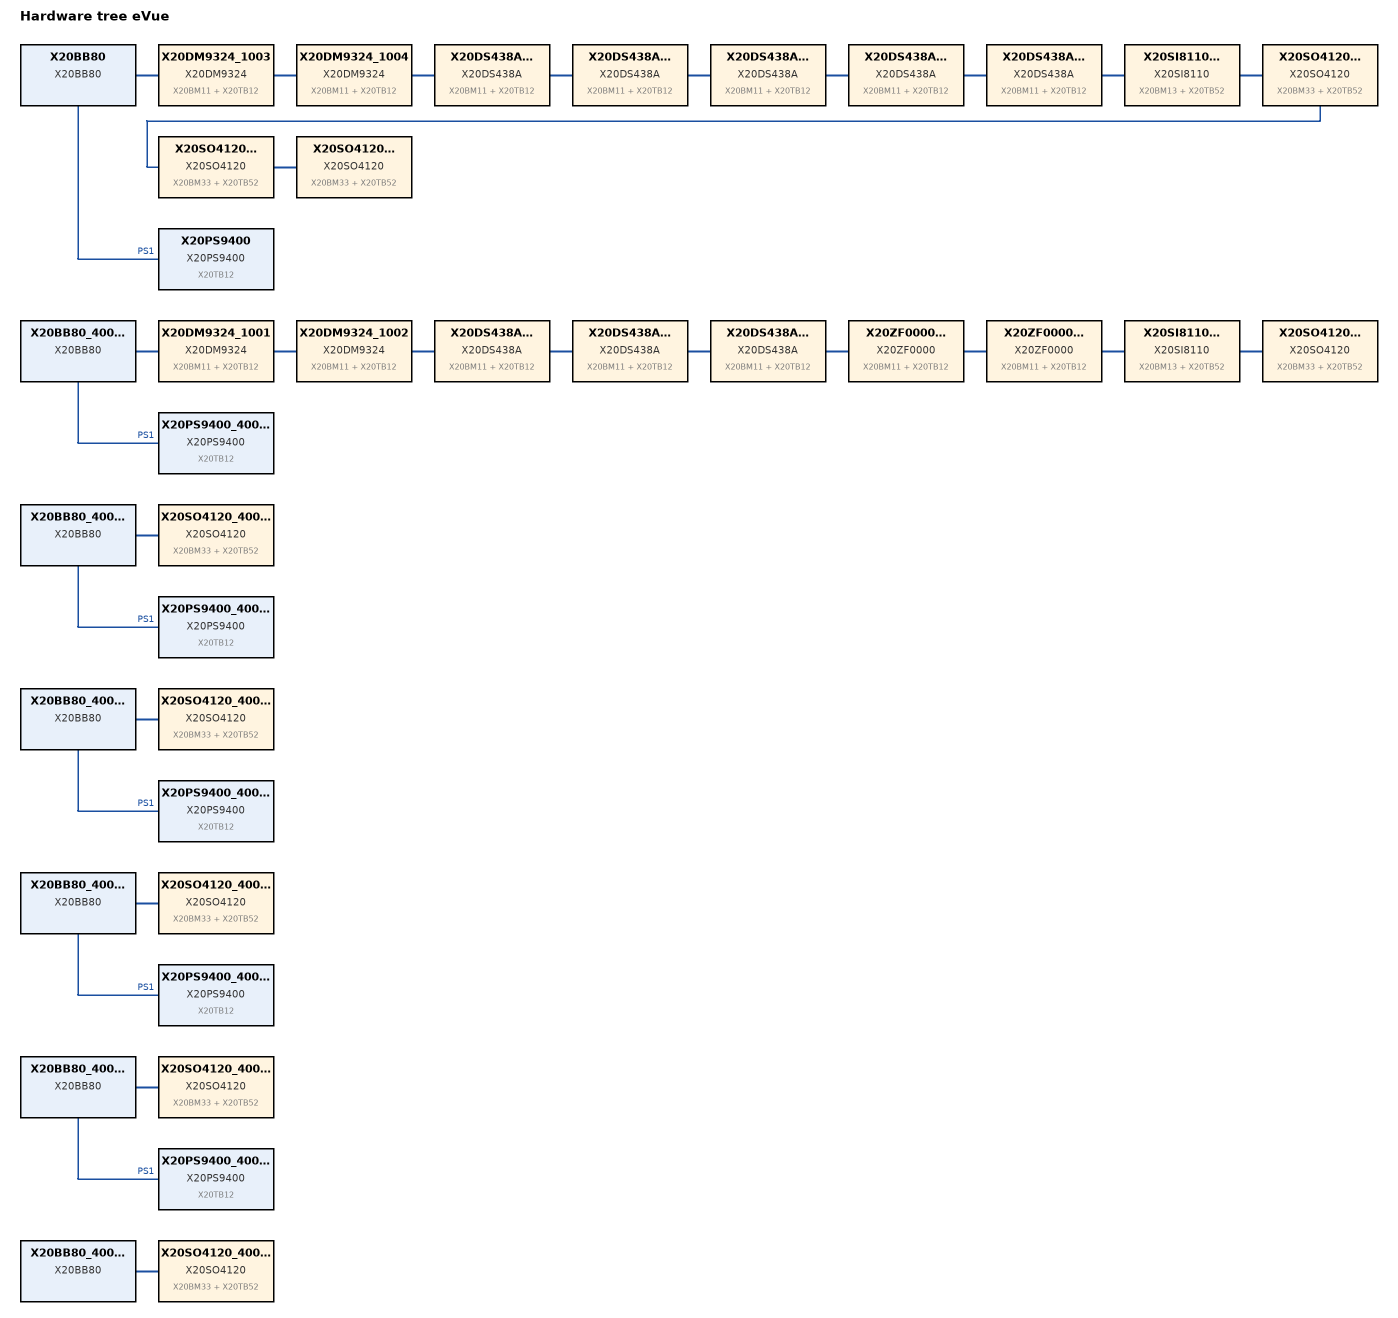
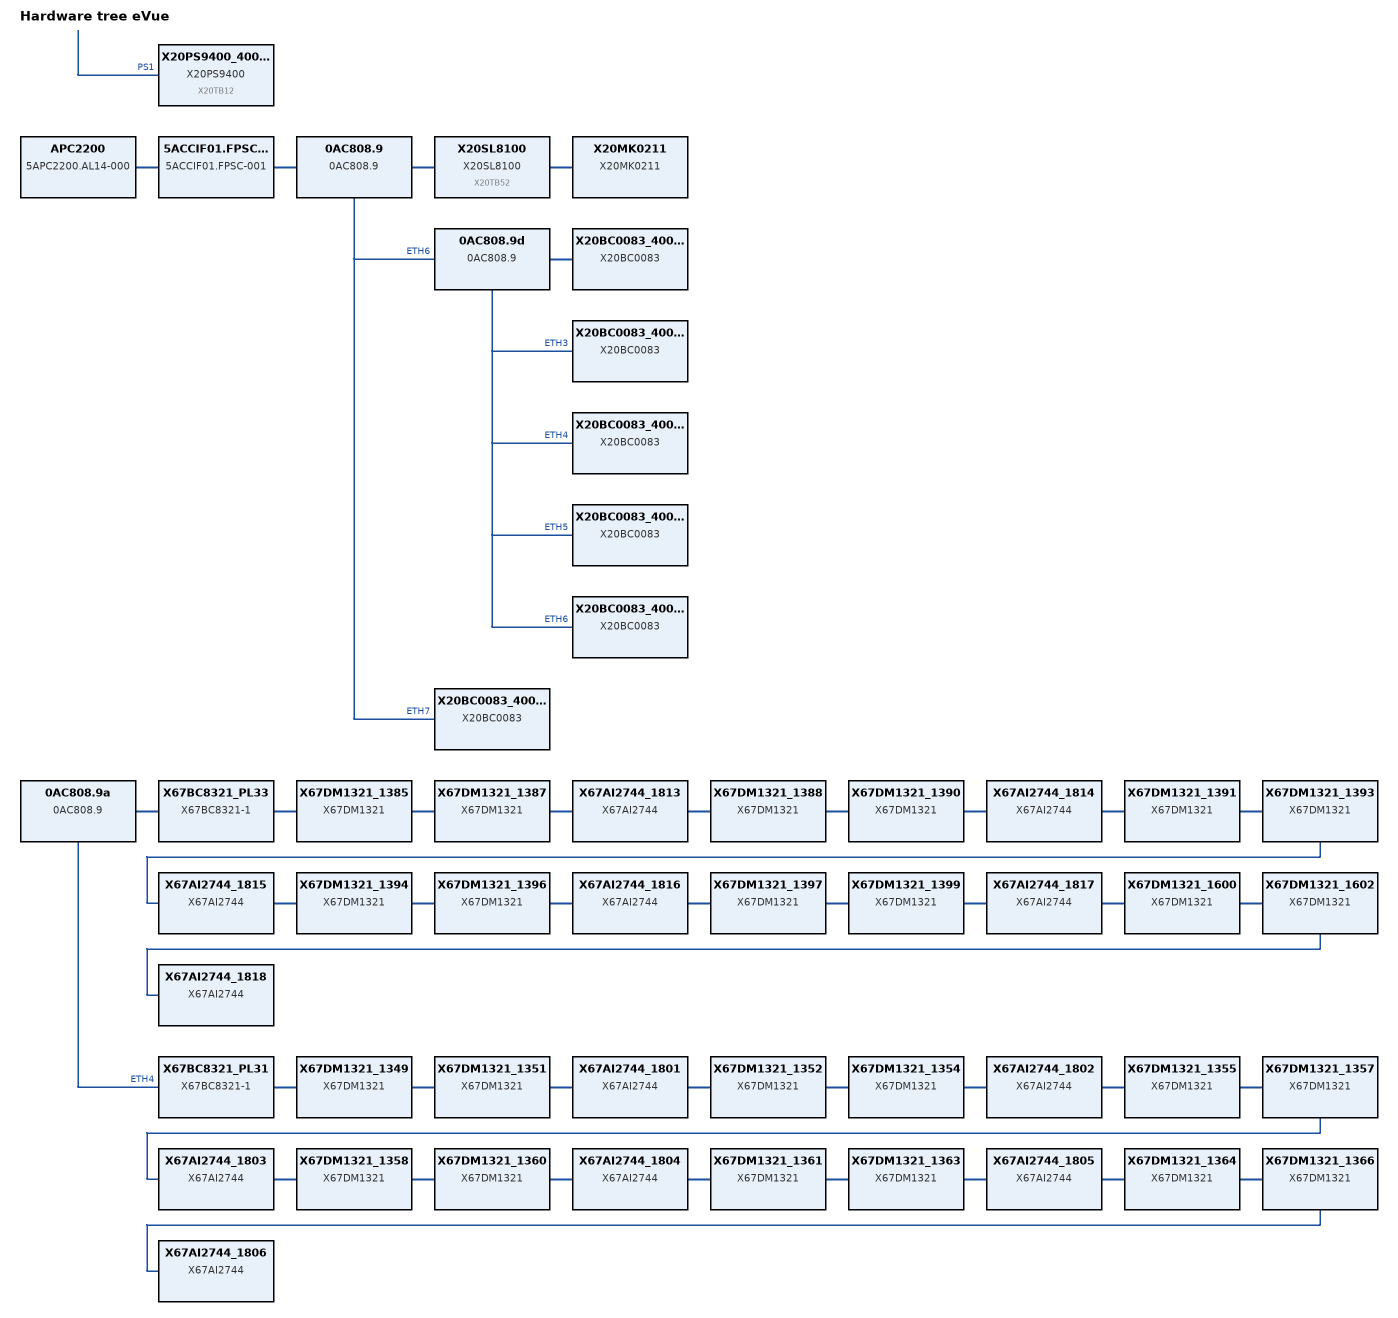
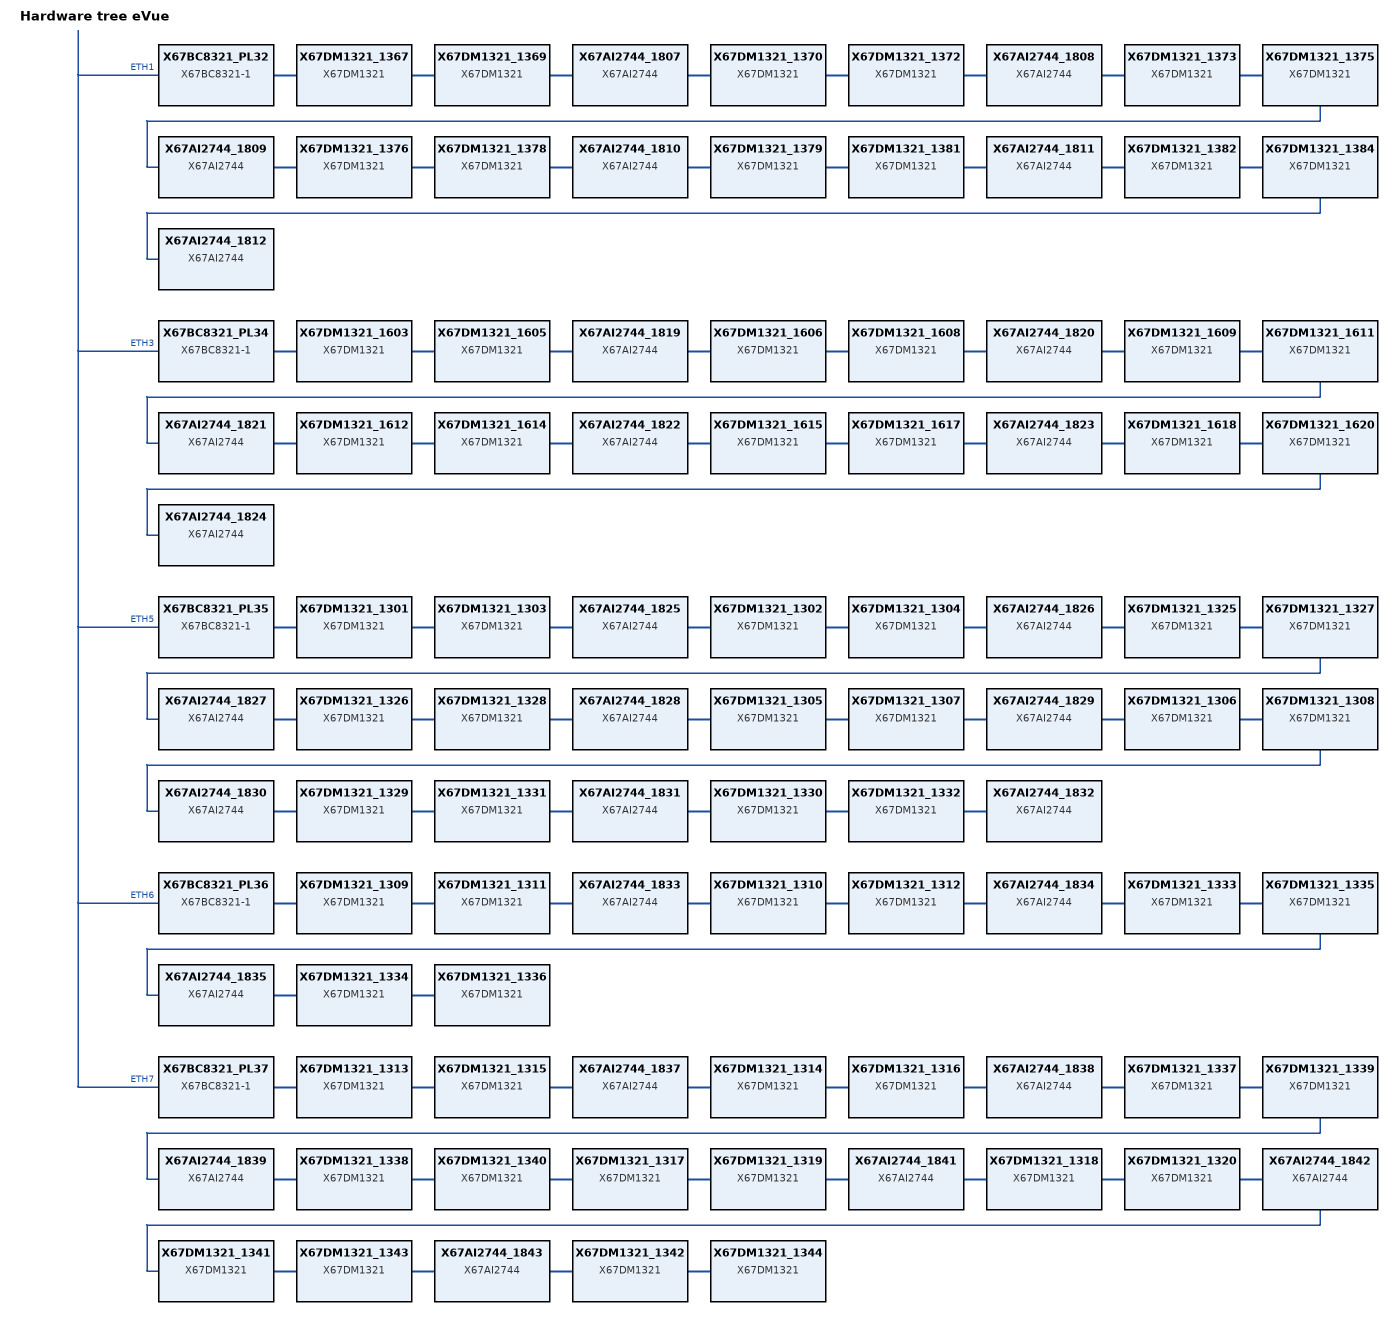
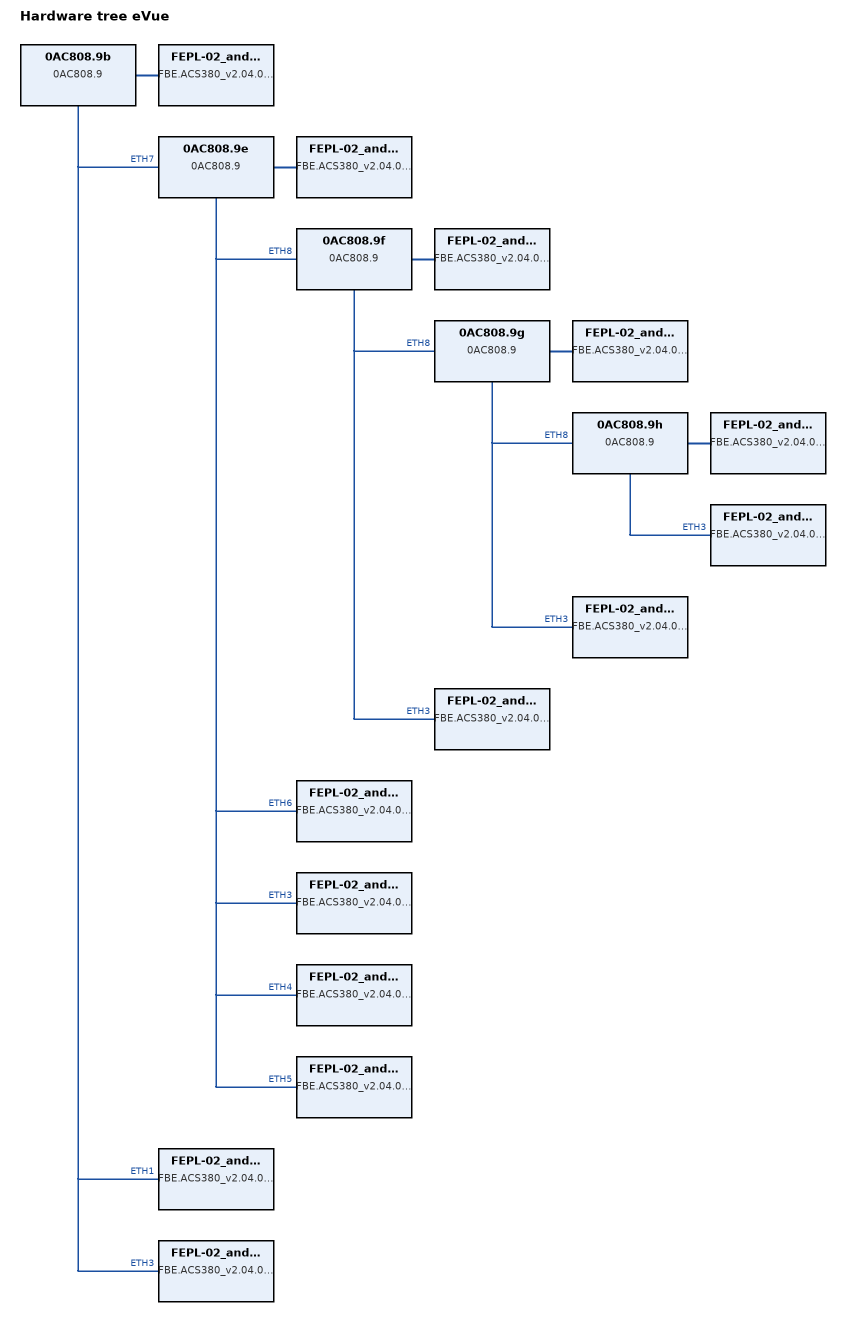
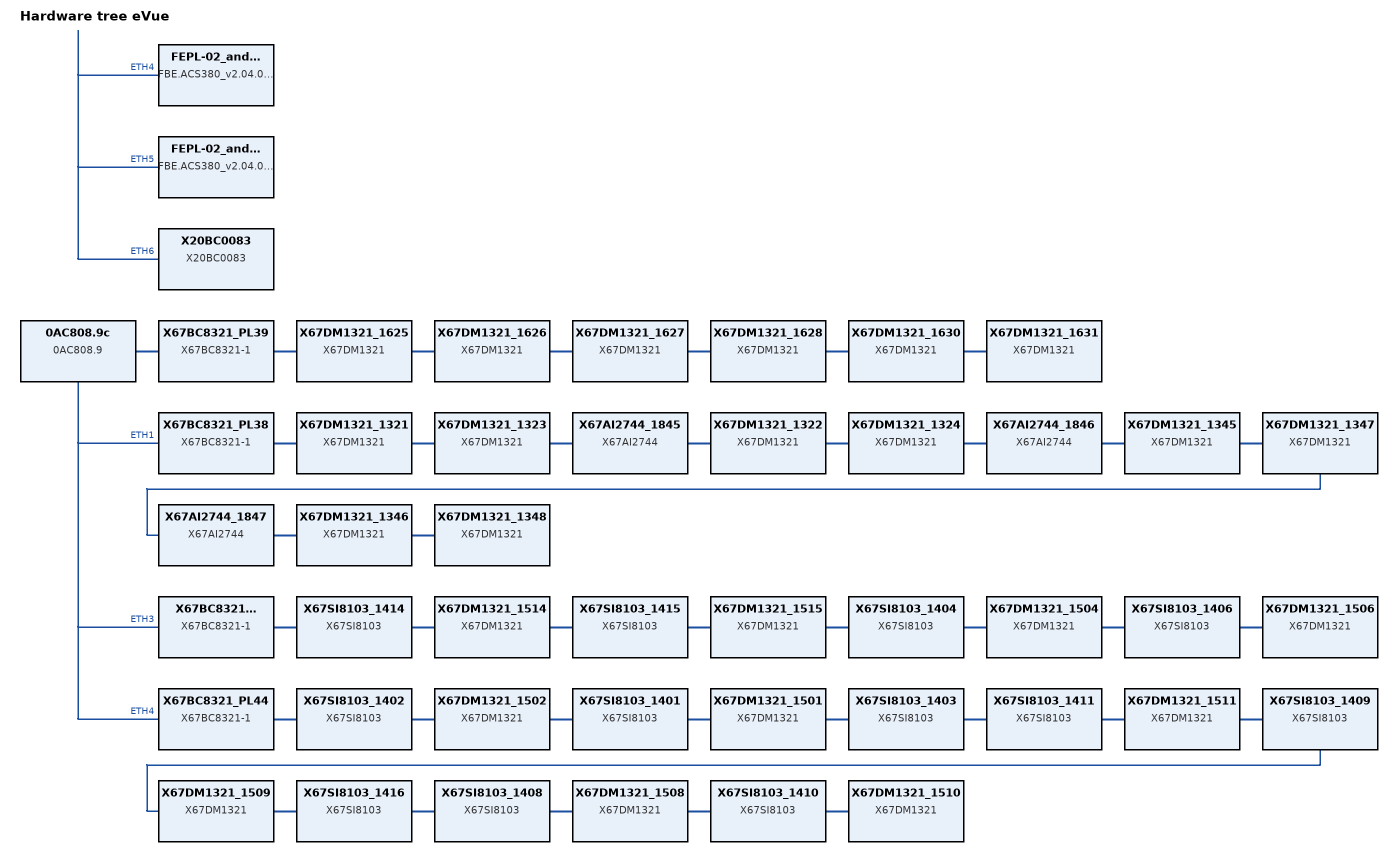
```
0AC808.9 : 0AC808.9 v1.0.0.0  [ETH1 -> 5ACCIF01.FPSC-001.IF1 [Cable Type=PowerlinkCable, Length=10, Version=1.0.0.3]; ETH2 -> X20SL8100.PLK1 [Cable Type=PowerlinkCable, Length=10, Version=1.0.0.3]; ETH4 -> 0AC808.9c.ETH8 [Cable Type=PowerlinkCable, Length=10, Version=1.0.0.3]; ETH6 -> 0AC808.9d.ETH1 [Cable Type=PowerlinkCable, Length=10, Version=1.0.0.3]; ETH7 -> X20BC0083_400_MC01.PLK1 [Cable Type=PowerlinkCable, Length=10, Version=1.0.0.3]; ETH8 -> 0AC808.9a.ETH8 [Cable Type=PowerlinkCable, Length=10, Version=1.0.0.3]]
0AC808.9a : 0AC808.9 v1.0.0.0  [ETH1 -> X67BC8321_PL32.PLK1 [Cable Type=PowerlinkCable, Length=10, Version=1.0.0.3]; ETH2 -> X67BC8321_PL33.PLK1 [Cable Type=PowerlinkCable, Length=10, Version=1.0.0.3]; ETH3 -> X67BC8321_PL34.PLK1 [Cable Type=PowerlinkCable, Length=10, Version=1.0.0.3]; ETH4 -> X67BC8321_PL31.PLK1 [Cable Type=PowerlinkCable, Length=10, Version=1.0.0.3]; ETH5 -> X67BC8321_PL35.PLK1 [Cable Type=PowerlinkCable, Length=10, Version=1.0.0.3]; ETH6 -> X67BC8321_PL36.PLK1 [Cable Type=PowerlinkCable, Length=10, Version=1.0.0.3]; ETH7 -> X67BC8321_PL37.PLK1 [Cable Type=PowerlinkCable, Length=10, Version=1.0.0.3]; ETH8 -> 0AC808.9.ETH8 [Cable Type=PowerlinkCable, Length=10, Version=1.0.0.3]]
0AC808.9b : 0AC808.9 v1.0.0.0  [ETH1 -> FEPL-02_and_ACS380_STB1.PLK1 [Cable Type=PowerlinkCable, Length=10, Version=1.0.0.3]; ETH2 -> FEPL-02_and_ACS380_STB2.PLK1 [Cable Type=PowerlinkCable, Length=10, Version=1.0.0.3]; ETH3 -> FEPL-02_and_ACS380_STB5.PLK1 [Cable Type=PowerlinkCable, Length=10, Version=1.0.0.3]; ETH4 -> FEPL-02_and_ACS380_STB6.PLK1 [Cable Type=PowerlinkCable, Length=10, Version=1.0.0.3]; ETH5 -> FEPL-02_and_ACS380_STB7.PLK1 [Cable Type=PowerlinkCable, Length=10, Version=1.0.0.3]; ETH6 -> X20BC0083.PLK1 [Cable Type=PowerlinkCable, Length=10, Version=1.0.0.3]; ETH7 -> 0AC808.9e.ETH1 [Cable Type=PowerlinkCable, Length=10, Version=1.0.0.3]; ETH8 -> 0AC808.9d.ETH8 [Cable Type=PowerlinkCable, Length=10, Version=1.0.0.3]]
0AC808.9c : 0AC808.9 v1.0.0.0  [ETH1 -> X67BC8321_PL38.PLK1 [Cable Type=PowerlinkCable, Length=10, Version=1.0.0.3]; ETH2 -> X67BC8321_PL39.PLK1 [Cable Type=PowerlinkCable, Length=10, Version=1.0.0.3]; ETH3 -> X67BC8321_PL43_S.PLK1 [Cable Type=PowerlinkCable, Length=10, Version=1.0.0.3]; ETH4 -> X67BC8321_PL44.PLK1 [Cable Type=PowerlinkCable, Length=10, Version=1.0.0.3]; ETH8 -> 0AC808.9.ETH4 [Cable Type=PowerlinkCable, Length=10, Version=1.0.0.3]]
0AC808.9d : 0AC808.9 v1.0.0.0  [ETH1 -> 0AC808.9.ETH6 [Cable Type=PowerlinkCable, Length=10, Version=1.0.0.3]; ETH2 -> X20BC0083_400_SC01.PLK1 [Cable Type=PowerlinkCable, Length=10, Version=1.0.0.3]; ETH3 -> X20BC0083_400_SC02.PLK1 [Cable Type=PowerlinkCable, Length=10, Version=1.0.0.3]; ETH4 -> X20BC0083_400_SC03.PLK1 [Cable Type=PowerlinkCable, Length=10, Version=1.0.0.3]; ETH5 -> X20BC0083_400_SC04.PLK1 [Cable Type=PowerlinkCable, Length=10, Version=1.0.0.3]; ETH6 -> X20BC0083_400_SC05.PLK1 [Cable Type=PowerlinkCable, Length=10, Version=1.0.0.3]; ETH8 -> 0AC808.9b.ETH8 [Cable Type=PowerlinkCable, Length=10, Version=1.0.0.3]]
0AC808.9e : 0AC808.9 v1.0.0.0  [ETH1 -> 0AC808.9b.ETH7 [Cable Type=PowerlinkCable, Length=10, Version=1.0.0.3]; ETH2 -> FEPL-02_and_ACS380_STB3.PLK1 [Cable Type=PowerlinkCable, Length=10, Version=1.0.0.3]; ETH3 -> FEPL-02_and_ACS380_STB4.PLK1 [Cable Type=PowerlinkCable, Length=10, Version=1.0.0.3]; ETH4 -> FEPL-02_and_ACS380_STB8.PLK1 [Cable Type=PowerlinkCable, Length=10, Version=1.0.0.3]; ETH5 -> FEPL-02_and_ACS380_STB9.PLK1 [Cable Type=PowerlinkCable, Length=10, Version=1.0.0.3]; ETH6 -> FEPL-02_and_ACS380_STB10.PLK1 [Cable Type=PowerlinkCable, Length=10, Version=1.0.0.3]; ETH8 -> 0AC808.9f.ETH1 [Cable Type=PowerlinkCable, Length=10, Version=1.0.0.3]]
0AC808.9f : 0AC808.9 v1.0.0.0  [ETH1 -> 0AC808.9e.ETH8 [Cable Type=PowerlinkCable, Length=10, Version=1.0.0.3]; ETH2 -> FEPL-02_and_ACS380_SB1.PLK1 [Cable Type=PowerlinkCable, Length=10, Version=1.0.0.3]; ETH3 -> FEPL-02_and_ACS380_SB2.PLK1 [Cable Type=PowerlinkCable, Length=10, Version=1.0.0.3]; ETH8 -> 0AC808.9g.ETH1 [Cable Type=PowerlinkCable, Length=10, Version=1.0.0.3]]
0AC808.9g : 0AC808.9 v1.0.0.0  [ETH1 -> 0AC808.9f.ETH8 [Cable Type=PowerlinkCable, Length=10, Version=1.0.0.3]; ETH2 -> FEPL-02_and_ACS380_SB3.PLK1 [Cable Type=PowerlinkCable, Length=10, Version=1.0.0.3]; ETH3 -> FEPL-02_and_ACS380_SB4.PLK1 [Cable Type=PowerlinkCable, Length=10, Version=1.0.0.3]; ETH8 -> 0AC808.9h.ETH1 [Cable Type=PowerlinkCable, Length=10, Version=1.0.0.3]]
0AC808.9h : 0AC808.9 v1.0.0.0  [ETH1 -> 0AC808.9g.ETH8 [Cable Type=PowerlinkCable, Length=10, Version=1.0.0.3]; ETH2 -> FEPL-02_and_ACS380_STB11.PLK1 [Cable Type=PowerlinkCable, Length=10, Version=1.0.0.3]; ETH3 -> FEPL-02_and_ACS380_STB12.PLK1 [Cable Type=PowerlinkCable, Length=10, Version=1.0.0.3]]
5ACCIF01.FPSC-001 : 5ACCIF01.FPSC-001 v1.8.1.0  [SL -> APC2200.SL1]
  Connector IF1:
    MtuSize  // *Increase packet size
    DNAConfiguration = manual
    AsyncTimeout = 300
    InternetAddress = 192.168.201.240  // * Static IP -- Must be 200 + PLC ip end -- Ie. 10.8.12.31  -- EPL = 192.168.201.240
    SubnetMask = 255.255.255.0
  Connector IF3:
    Baudrate = 250000
    ActivateCanOpen = 1
    pcannodeid = 2
    pnmtstartup_bit3 = 1
    pnmtstartup_maximumbootuptime = 20
    pheartbeat_producertime = 500
    pactivatesync = 1
    pcycleperiod = 10000
    pwindowlength = 10000
APC2200 : 5APC2200.AL14-000 v2.0.1.0
  Connector IF3:
    AssignedOperatingSystem = ARemb
    ActivateDevice = 1
    Mode = Manual
    InternetAddress = 10.8.12.31
    SubnetMask = 255.255.240.0
    InaNodeNumber = 0
  Connector IF4:
    AssignedOperatingSystem = ARemb
    ActivateDevice = 1
  Connector IF5:
    AssignedOperatingSystem = ARemb
  Connector IF6:
    AssignedOperatingSystem = ARemb
  ConfigurationID = 8245
  UserRamDevice = PCI.1.PPC21xx.SRAM
  UserRamSize = 400000
  RemMemDevice = PCI.1.PPC21xx.SRAM
  RemMemSize = 108000
  PermanentPvSize = 30000
  RemanentGlobalPvSize = 12000
  VolatileGlobalPvSize = 5000000
  EnableUsbRemoteInstall = 1
  EnableCfRemoteInstall = 1
  Cyclic1Duration = 1000
  Cyclic1Tolerance = 2000
  Cyclic2Duration = 12000
  Cyclic2Tolerance = 12000
  Cyclic3Duration = 12000
  Cyclic3Tolerance = 12000
  Cyclic4Duration = 12000
  Cyclic4Tolerance = 12000
  Cyclic5Duration = 12000
  Cyclic5Tolerance = 12000
  Cyclic6Duration = 54000
  Cyclic6Tolerance = 54000
  Cyclic7Duration = 102000
  Cyclic7Tolerance = 102000
  Cyclic8Duration = 12000
  FileDevice1
  FileDeviceName1 = user
  FileDevicePath1 = F:/
  ActivateDaylightSavingTime = 1
  ActivateSntp = 1
  SntpcServAddr1 = 10.8.15.254
  SntpcServAddr2 = 10.8.4.220
  EthernetHostName = SupertrackPLC
  EthernetDefaultGateway = 10.8.15.254
  FtpUser1
  FtpUsername1 = admin
  FtpUserPassword1 = BySUEieH3gX7lWqprIraeTLnjrwkiLwh2+z9OmyZ02E=  // admin
  FtpUserSalt1 = ywni0ciN
  FTPAccessRight1 = 0
  ActivateOpcUa = 1
  OpcUaInformationModels_PV_Version = 1
  Cyclic8Tolerance = 30000000
FEPL-02_and_ACS380_SB1 : FBE.ACS380_v2.04.0.3_FEPL-02_1.0_filerev1.0 vFFEPS10 (OrderNumber=FEPL-02 and ACS380)  [PLK1 -> 0AC808.9f.ETH2 (NodeNumber=131) [Cable Type=PowerlinkCable, Length=10, Version=1.0.0.3]]
  Supervision = off
  p2203_direction = ro
  p6040_direction = wo
  p6041_direction = ro
  p6042_direction = wo
  p6044_direction = ro
  p4001s07_direction = ro
  p4001s0A_direction = ro
FEPL-02_and_ACS380_SB2 : FBE.ACS380_v2.04.0.3_FEPL-02_1.0_filerev1.0 vFFEPS10 (OrderNumber=FEPL-02 and ACS380)  [PLK1 -> 0AC808.9f.ETH3 (NodeNumber=132) [Cable Type=PowerlinkCable, Length=10, Version=1.0.0.3]]
  Supervision = off
  p2203_direction = ro
  p6040_direction = wo
  p6041_direction = ro
  p6042_direction = wo
  p6044_direction = ro
  p4001s07_direction = ro
  p4001s0A_direction = ro
FEPL-02_and_ACS380_SB3 : FBE.ACS380_v2.04.0.3_FEPL-02_1.0_filerev1.0 vFFEPS10 (OrderNumber=FEPL-02 and ACS380)  [PLK1 -> 0AC808.9g.ETH2 (NodeNumber=141) [Cable Type=PowerlinkCable, Length=10, Version=1.0.0.3]]
  Supervision = off
  p2203_direction = ro
  p6040_direction = wo
  p6041_direction = ro
  p6042_direction = wo
  p6044_direction = ro
  p4001s07_direction = ro
  p4001s0A_direction = ro
FEPL-02_and_ACS380_SB4 : FBE.ACS380_v2.04.0.3_FEPL-02_1.0_filerev1.0 vFFEPS10 (OrderNumber=FEPL-02 and ACS380)  [PLK1 -> 0AC808.9g.ETH3 (NodeNumber=142) [Cable Type=PowerlinkCable, Length=10, Version=1.0.0.3]]
  Supervision = off
  p2203_direction = ro
  p6040_direction = wo
  p6041_direction = ro
  p6042_direction = wo
  p6044_direction = ro
  p4001s07_direction = ro
  p4001s0A_direction = ro
FEPL-02_and_ACS380_STB1 : FBE.ACS380_v2.04.0.3_FEPL-02_1.0_filerev1.0 vFFEPS10 (OrderNumber=FEPL-02 and ACS380)  [PLK1 -> 0AC808.9b.ETH1 (NodeNumber=111) [Cable Type=PowerlinkCable, Length=10, Version=1.0.0.3]]
  Supervision = off
  p2203_direction = ro
  p6040_direction = wo
  p6041_direction = ro
  p6042_direction = wo
  p6044_direction = ro
  p4001s07_direction = ro
  p4001s0A_direction = ro
FEPL-02_and_ACS380_STB10 : FBE.ACS380_v2.04.0.3_FEPL-02_1.0_filerev1.0 vFFEPS10 (OrderNumber=FEPL-02 and ACS380)  [PLK1 -> 0AC808.9e.ETH6 (NodeNumber=125) [Cable Type=PowerlinkCable, Length=10, Version=1.0.0.3]]
  Supervision = off
  p2203_direction = ro
  p6040_direction = wo
  p6041_direction = ro
  p6042_direction = wo
  p6044_direction = ro
  p4001s07_direction = ro
  p4001s0A_direction = ro
FEPL-02_and_ACS380_STB11 : FBE.ACS380_v2.04.0.3_FEPL-02_1.0_filerev1.0 vFFEPS10 (OrderNumber=FEPL-02 and ACS380)  [PLK1 -> 0AC808.9h.ETH2 (NodeNumber=151) [Cable Type=PowerlinkCable, Length=10, Version=1.0.0.3]]
  Supervision = off
  p2203_direction = ro
  p6040_direction = wo
  p6041_direction = ro
  p6042_direction = wo
  p6044_direction = ro
  p4001s07_direction = ro
  p4001s0A_direction = ro
FEPL-02_and_ACS380_STB12 : FBE.ACS380_v2.04.0.3_FEPL-02_1.0_filerev1.0 vFFEPS10 (OrderNumber=FEPL-02 and ACS380)  [PLK1 -> 0AC808.9h.ETH3 (NodeNumber=152) [Cable Type=PowerlinkCable, Length=10, Version=1.0.0.3]]
  Supervision = off
  p2203_direction = ro
  p6040_direction = wo
  p6041_direction = ro
  p6042_direction = wo
  p6044_direction = ro
  p4001s07_direction = ro
  p4001s0A_direction = ro
FEPL-02_and_ACS380_STB2 : FBE.ACS380_v2.04.0.3_FEPL-02_1.0_filerev1.0 vFFEPS10 (OrderNumber=FEPL-02 and ACS380)  [PLK1 -> 0AC808.9b.ETH2 (NodeNumber=112) [Cable Type=PowerlinkCable, Length=10, Version=1.0.0.3]]
  Supervision = off
  p2203_direction = ro
  p6040_direction = wo
  p6041_direction = ro
  p6042_direction = wo
  p6044_direction = ro
  p4001s07_direction = ro
  p4001s0A_direction = ro
FEPL-02_and_ACS380_STB3 : FBE.ACS380_v2.04.0.3_FEPL-02_1.0_filerev1.0 vFFEPS10 (OrderNumber=FEPL-02 and ACS380)  [PLK1 -> 0AC808.9e.ETH2 (NodeNumber=121) [Cable Type=PowerlinkCable, Length=10, Version=1.0.0.3]]
  Supervision = off
  p2203_direction = ro
  p6040_direction = wo
  p6041_direction = ro
  p6042_direction = wo
  p6044_direction = ro
  p4001s07_direction = ro
  p4001s0A_direction = ro
FEPL-02_and_ACS380_STB4 : FBE.ACS380_v2.04.0.3_FEPL-02_1.0_filerev1.0 vFFEPS10 (OrderNumber=FEPL-02 and ACS380)  [PLK1 -> 0AC808.9e.ETH3 (NodeNumber=122) [Cable Type=PowerlinkCable, Length=10, Version=1.0.0.3]]
  Supervision = off
  p2203_direction = ro
  p6040_direction = wo
  p6041_direction = ro
  p6042_direction = wo
  p6044_direction = ro
  p4001s07_direction = ro
  p4001s0A_direction = ro
FEPL-02_and_ACS380_STB5 : FBE.ACS380_v2.04.0.3_FEPL-02_1.0_filerev1.0 vFFEPS10 (OrderNumber=FEPL-02 and ACS380)  [PLK1 -> 0AC808.9b.ETH3 (NodeNumber=113) [Cable Type=PowerlinkCable, Length=10, Version=1.0.0.3]]
  Supervision = off
  p2203_direction = ro
  p6040_direction = wo
  p6041_direction = ro
  p6042_direction = wo
  p6044_direction = ro
  p4001s07_direction = ro
  p4001s0A_direction = ro
FEPL-02_and_ACS380_STB6 : FBE.ACS380_v2.04.0.3_FEPL-02_1.0_filerev1.0 vFFEPS10 (OrderNumber=FEPL-02 and ACS380)  [PLK1 -> 0AC808.9b.ETH4 (NodeNumber=114) [Cable Type=PowerlinkCable, Length=10, Version=1.0.0.3]]
  Supervision = off
  p2203_direction = ro
  p6040_direction = wo
  p6041_direction = ro
  p6042_direction = wo
  p6044_direction = ro
  p4001s07_direction = ro
  p4001s0A_direction = ro
FEPL-02_and_ACS380_STB7 : FBE.ACS380_v2.04.0.3_FEPL-02_1.0_filerev1.0 vFFEPS10 (OrderNumber=FEPL-02 and ACS380)  [PLK1 -> 0AC808.9b.ETH5 (NodeNumber=115) [Cable Type=PowerlinkCable, Length=10, Version=1.0.0.3]]
  Supervision = off
  p2203_direction = ro
  p6040_direction = wo
  p6041_direction = ro
  p6042_direction = wo
  p6044_direction = ro
  p4001s07_direction = ro
  p4001s0A_direction = ro
FEPL-02_and_ACS380_STB8 : FBE.ACS380_v2.04.0.3_FEPL-02_1.0_filerev1.0 vFFEPS10 (OrderNumber=FEPL-02 and ACS380)  [PLK1 -> 0AC808.9e.ETH4 (NodeNumber=123) [Cable Type=PowerlinkCable, Length=10, Version=1.0.0.3]]
  Supervision = off
  p2203_direction = ro
  p6040_direction = wo
  p6041_direction = ro
  p6042_direction = wo
  p6044_direction = ro
  p4001s07_direction = ro
  p4001s0A_direction = ro
FEPL-02_and_ACS380_STB9 : FBE.ACS380_v2.04.0.3_FEPL-02_1.0_filerev1.0 vFFEPS10 (OrderNumber=FEPL-02 and ACS380)  [PLK1 -> 0AC808.9e.ETH5 (NodeNumber=124) [Cable Type=PowerlinkCable, Length=10, Version=1.0.0.3]]
  Supervision = off
  p2203_direction = ro
  p6040_direction = wo
  p6041_direction = ro
  p6042_direction = wo
  p6044_direction = ro
  p4001s07_direction = ro
  p4001s0A_direction = ro
X20BB80 : X20BB80 v1.0.2.0
X20BB80_400_MC01 : X20BB80 v1.0.2.0
X20BB80_400_SC01 : X20BB80 v1.0.2.0
X20BB80_400_SC02 : X20BB80 v1.0.2.0
X20BB80_400_SC03 : X20BB80 v1.0.2.0
X20BB80_400_SC04 : X20BB80 v1.0.2.0
X20BB80_400_SC05 : X20BB80 v1.0.2.0
X20BC0083 : X20BC0083 v2.11.1.0  [PLK1 -> 0AC808.9b.ETH6 (NodeNumber=22) [Cable Type=PowerlinkCable, Length=10, Version=1.0.0.3]; SL -> X20BB80.SL1]
  Supervision = off
X20BC0083_400_MC01 : X20BC0083 v2.11.1.0  [PLK1 -> 0AC808.9.ETH7 (NodeNumber=21) [Cable Type=PowerlinkCable, Length=10, Version=1.0.0.3]; SL -> X20BB80_400_MC01.SL1]
  Supervision = off
X20BC0083_400_SC01 : X20BC0083 v2.11.1.0  [PLK1 -> 0AC808.9d.ETH2 (NodeNumber=110) [Cable Type=PowerlinkCable, Length=10, Version=1.0.0.3]; SL -> X20BB80_400_SC01.SL1]
  Supervision = off
X20BC0083_400_SC02 : X20BC0083 v2.11.1.0  [PLK1 -> 0AC808.9d.ETH3 (NodeNumber=120) [Cable Type=PowerlinkCable, Length=10, Version=1.0.0.3]; SL -> X20BB80_400_SC02.SL1]
  Supervision = off
X20BC0083_400_SC03 : X20BC0083 v2.11.1.0  [PLK1 -> 0AC808.9d.ETH4 (NodeNumber=130) [Cable Type=PowerlinkCable, Length=10, Version=1.0.0.3]; SL -> X20BB80_400_SC03.SL1]
  Supervision = off
X20BC0083_400_SC04 : X20BC0083 v2.11.1.0  [PLK1 -> 0AC808.9d.ETH5 (NodeNumber=140) [Cable Type=PowerlinkCable, Length=10, Version=1.0.0.3]; SL -> X20BB80_400_SC04.SL1]
  Supervision = off
X20BC0083_400_SC05 : X20BC0083 v2.11.1.0  [PLK1 -> 0AC808.9d.ETH6 (NodeNumber=150) [Cable Type=PowerlinkCable, Length=10, Version=1.0.0.3]; SL -> X20BB80_400_SC05.SL1]
  Supervision = off
X20BM11 : X20BM11 v1.0.0.1  [X2X1 -> X20BB80_400_MC01.IF1]
X20BM11a : X20BM11 v1.0.0.1  [X2X1 -> X20BM11.X2X2]
X20BM11b : X20BM11 v1.0.0.1  [X2X1 -> X20BM11a.X2X2]
X20BM11c : X20BM11 v1.0.0.1  [X2X1 -> X20BM11d.X2X2]
X20BM11d : X20BM11 v1.0.0.1  [X2X1 -> X20BM11f.X2X2]
X20BM11e : X20BM11 v1.0.0.1  [X2X1 -> X20BM11c.X2X2]
X20BM11f : X20BM11 v1.0.0.1  [X2X1 -> X20BM11b.X2X2]
X20BM11g : X20BM11 v1.0.0.1  [X2X1 -> X20BB80.IF1]
X20BM11h : X20BM11 v1.0.0.1  [X2X1 -> X20BM11g.X2X2]
X20BM11i : X20BM11 v1.0.0.1  [X2X1 -> X20BM11h.X2X2]
X20BM11j : X20BM11 v1.0.0.1  [X2X1 -> X20BM11i.X2X2]
X20BM11k : X20BM11 v1.0.0.1  [X2X1 -> X20BM11j.X2X2]
X20BM11l : X20BM11 v1.0.0.1  [X2X1 -> X20BM11k.X2X2]
X20BM11m : X20BM11 v1.0.0.1  [X2X1 -> X20BM11l.X2X2]
X20BM13 : X20BM13 v1.0.0.6  [X2X1 -> X20BM11e.X2X2]
X20BM13a : X20BM13 v1.0.0.6  [X2X1 -> X20BM11m.X2X2]
X20BM33 : X20BM33 v1.0.0.6  [X2X1 -> X20BM13.X2X2]
X20BM33a : X20BM33 v1.0.0.6  [X2X1 -> X20BB80_400_SC02.IF1]
X20BM33b : X20BM33 v1.0.0.6  [X2X1 -> X20BB80_400_SC03.IF1]
X20BM33c : X20BM33 v1.0.0.6  [X2X1 -> X20BB80_400_SC04.IF1]
X20BM33d : X20BM33 v1.0.0.6  [X2X1 -> X20BB80_400_SC01.IF1]
X20BM33e : X20BM33 v1.0.0.6  [X2X1 -> X20BB80_400_SC05.IF1]
X20BM33f : X20BM33 v1.0.0.6  [X2X1 -> X20BM13a.X2X2]
X20BM33g : X20BM33 v1.0.0.6  [X2X1 -> X20BM33f.X2X2]
X20BM33h : X20BM33 v1.0.0.6  [X2X1 -> X20BM33g.X2X2]
X20DM9324_1001 : X20DM9324 v1.1.0.0  [SS1 -> X20TB12a.SS; SL -> X20BM11.SL1]
  Supervision = off
X20DM9324_1002 : X20DM9324 v1.1.0.0  [SS1 -> X20TB12.SS; SL -> X20BM11a.SL1]
  Supervision = off
X20DM9324_1003 : X20DM9324 v1.1.0.0  [SS1 -> X20TB12n.SS; SL -> X20BM11g.SL1]
  Supervision = off
X20DM9324_1004 : X20DM9324 v1.1.0.0  [SS1 -> X20TB12o.SS; SL -> X20BM11h.SL1]
  Supervision = off
X20DS438A_MC01_K103 : X20DS438A v2.2.0.0  [SS1 -> X20TB12c.SS; SL -> X20BM11b.SL1]
  DtmRef = FBD.BRIOLinkModuleDTM.DTMCore.X20DS438A
  DtmId = ebcb262e-d1f2-4f06-8305-bc88af423653
  CommDtmId = 00afcaaa-3871-4494-8c19-850a53e1ac49
  RequiresDTMBuild = true
  ConfigFile = Communication.dtm
  ConfigModule = asiol1
  Supervision = off
  OperatingMode01 = Operate
  OperatingMode02 = Operate
  OperatingMode03 = Operate
X20DS438A_MC01_K104 : X20DS438A v2.2.0.0  [SS1 -> X20TB12h.SS; SL -> X20BM11f.SL1]
  DtmRef = FBD.BRIOLinkModuleDTM.DTMCore.X20DS438A
  DtmId = 471367e8-93ce-4547-a931-5ad010e9f84c
  CommDtmId = 00afcaaa-3871-4494-8c19-850a53e1ac49
  RequiresDTMBuild = true
  ConfigFile = Communication.dtm
  ConfigModule = asiol3
  Supervision = off
  OperatingMode01 = Operate
  OperatingMode02 = Operate
  OperatingMode03 = Operate
X20DS438A_MC01_K105 : X20DS438A v2.2.0.0  [SS1 -> X20TB12e.SS; SL -> X20BM11d.SL1]
  DtmRef = FBD.BRIOLinkModuleDTM.DTMCore.X20DS438A
  DtmId = 4049e49e-fcbc-4ea6-8d89-ef98e0dd21ab
  CommDtmId = f6381c8e-a2e9-427a-8b33-d57985ec4dc6
  RequiresDTMBuild = true
  ConfigFile = Communication.dtm
  ConfigModule = asiol5
  Supervision = off
  OperatingMode01 = Operate
X20DS438A_MC02_Fuses_1 : X20DS438A v2.2.0.0  [SS1 -> X20TB12p.SS; SL -> X20BM11i.SL1]
  DtmRef = FBD.BRIOLinkModuleDTM.DTMCore.X20DS438A
  DtmId = 446c1e03-cea0-4ba5-8bc6-00e057ef7dbc
  CommDtmId = 5105a72f-3f3a-423d-add3-2a88fcfa15a0
  RequiresDTMBuild = true
  ConfigFile = Communication.dtm
  ConfigModule = asiol2
  Supervision = off
  OperatingMode01 = Operate
  OperatingMode02 = Operate
  OperatingMode03 = Operate
  OperatingMode04 = Operate
X20DS438A_MC02_Fuses_2 : X20DS438A v2.2.0.0  [SS1 -> X20TB12q.SS; SL -> X20BM11j.SL1]
  DtmRef = FBD.BRIOLinkModuleDTM.DTMCore.X20DS438A
  DtmId = 7f93e747-5eac-4250-902e-8361cfbb3373
  CommDtmId = 5105a72f-3f3a-423d-add3-2a88fcfa15a0
  RequiresDTMBuild = true
  ConfigFile = Communication.dtm
  ConfigModule = asiol4
  Supervision = off
  OperatingMode01 = Operate
  OperatingMode02 = Operate
  OperatingMode03 = Operate
X20DS438A_MC02_Fuses_3 : X20DS438A v2.2.0.0  [SS1 -> X20TB12r.SS; SL -> X20BM11k.SL1]
  DtmRef = FBD.BRIOLinkModuleDTM.DTMCore.X20DS438A
  DtmId = 910e90bf-845c-4123-a66a-7a431d3462a8
  CommDtmId = 5105a72f-3f3a-423d-add3-2a88fcfa15a0
  RequiresDTMBuild = true
  ConfigFile = Communication.dtm
  ConfigModule = asiol6
  Supervision = off
  OperatingMode01 = Operate
X20DS438A_MC02_Inclines_1 : X20DS438A v2.2.0.0  [SS1 -> X20TB12s.SS; SL -> X20BM11l.SL1]
  DtmRef = FBD.BRIOLinkModuleDTM.DTMCore.X20DS438A
  DtmId = 3b68baac-a41f-4b2b-a742-d8c170275c67
  CommDtmId = 5105a72f-3f3a-423d-add3-2a88fcfa15a0
  RequiresDTMBuild = true
  ConfigFile = Communication.dtm
  ConfigModule = asiol7
  Supervision = off
  OperatingMode01 = Operate
  PDI_Enable01 = octetArray_DPS
  PDI_OctetSizeDPS01 = 8byte
  PDO_Enable01 = variousTypes
  PDO_DataType01_1 = USINT
  PDO_DataType01_2 = USINT
  OperatingMode02 = Operate
  PDI_Enable02 = octetArray_DPS
  PDI_OctetSizeDPS02 = 8byte
  PDO_Enable02 = variousTypes
  PDO_DataType02_1 = USINT
  PDO_DataType02_2 = USINT
  OperatingMode03 = Operate
  PDI_Enable03 = octetArray_DPS
  PDI_OctetSizeDPS03 = 8byte
  PDO_Enable03 = variousTypes
  PDO_DataType03_1 = USINT
  PDO_DataType03_2 = USINT
  OperatingMode04 = Operate
  PDI_Enable04 = octetArray_DPS
  PDI_OctetSizeDPS04 = 8byte
  PDO_Enable04 = variousTypes
  PDO_DataType04_1 = USINT
  PDO_DataType04_2 = USINT
X20DS438A_MC02_Inclines_2 : X20DS438A v2.2.0.0  [SS1 -> X20TB12t.SS; SL -> X20BM11m.SL1]
  DtmRef = FBD.BRIOLinkModuleDTM.DTMCore.X20DS438A
  DtmId = 67f0ec63-a7b8-4edd-a572-cde922a25ead
  CommDtmId = 5105a72f-3f3a-423d-add3-2a88fcfa15a0
  RequiresDTMBuild = true
  ConfigFile = Communication.dtm
  ConfigModule = asiol8
  Supervision = off
  OperatingMode01 = Operate
  PDI_Enable01 = octetArray_DPS
  PDI_OctetSizeDPS01 = 8byte
  PDO_Enable01 = variousTypes
  PDO_DataType01_1 = USINT
  PDO_DataType01_2 = USINT
  OperatingMode02 = Operate
  PDI_Enable02 = octetArray_DPS
  PDI_OctetSizeDPS02 = 8byte
  PDO_Enable02 = variousTypes
  PDO_DataType02_1 = USINT
  PDO_DataType02_2 = USINT
  OperatingMode03 = Operate
  PDI_Enable03 = octetArray_DPS
  PDI_OctetSizeDPS03 = 8byte
  PDO_Enable03 = variousTypes
  PDO_DataType03_1 = USINT
  PDO_DataType03_2 = USINT
  OperatingMode04 = Operate
  PDI_Enable04 = octetArray_DPS
  PDI_OctetSizeDPS04 = 8byte
  PDO_Enable04 = variousTypes
  PDO_DataType04_1 = USINT
  PDO_DataType04_2 = USINT
X20MK0211 : X20MK0211 v1.0.0.3  [SL -> X20SL8100.SL1]
X20PS9400 : X20PS9400 v1.5.0.0  [SS1 -> X20TB12m.SS; PS -> X20BB80.PS1]
  Supervision = off
X20PS9400_400_MC01 : X20PS9400 v1.5.0.0  [SS1 -> X20TB12b.SS; PS -> X20BB80_400_MC01.PS1]
  Supervision = off
X20PS9400_400_SC01 : X20PS9400 v1.5.0.0  [SS1 -> X20TB12l.SS; PS -> X20BB80_400_SC01.PS1]
  Supervision = off
X20PS9400_400_SC02 : X20PS9400 v1.5.0.0  [SS1 -> X20TB12g.SS; PS -> X20BB80_400_SC02.PS1]
  Supervision = off
X20PS9400_400_SC03 : X20PS9400 v1.5.0.0  [SS1 -> X20TB12i.SS; PS -> X20BB80_400_SC03.PS1]
  Supervision = off
X20PS9400_400_SC04 : X20PS9400 v1.5.0.0  [SS1 -> X20TB12j.SS; PS -> X20BB80_400_SC04.PS1]
  Supervision = off
X20PS9400_400_SC05 : X20PS9400 v1.5.0.0  [SS1 -> X20TB12k.SS; PS -> X20BB80_400_SC05.PS1]
  Supervision = off
X20SI8110_MC01_K109 : X20SI8110 v2.3.1.0  [SS1 -> X20TB52.SS; SL -> X20BM13.SL1]
  Supervision = off
X20SI8110_MC02_K108 : X20SI8110 v2.3.1.0  [SS1 -> X20TB52g.SS; SL -> X20BM13a.SL1]
  Supervision = off
  SafeModuleID = 4
X20SL8100 : X20SL8100 v2.3.0.1  [PLK1 -> 0AC808.9.ETH2 (NodeNumber=239) [Cable Type=PowerlinkCable, Length=10, Version=1.0.0.3]; SS1 -> X20TB52c.SS]
  Supervision = off
  SafeProject = SafeLOGIC-1
  SafeDesigner = 4.1.3.3202125
  UnsafeOutputBOOLs = 0
  UnsafeOutputINTs = 1
  UnsafeOutputDINTs = 2
  UnsafeInputINTs = 30
X20SO4120_400_SC01 : X20SO4120 v2.2.1.0  [SS1 -> X20TB52h.SS; SL -> X20BM33d.SL1]
  Supervision = off
  SafeModuleID = 51
  DigitalOutput01 = viaSafeLOGIC
  DigitalOutput02 = viaSafeLOGIC
  DigitalOutput03 = viaSafeLOGIC
  DigitalOutput04 = viaSafeLOGIC
X20SO4120_400_SC02 : X20SO4120 v2.2.1.0  [SS1 -> X20TB52b.SS; SL -> X20BM33a.SL1]
  Supervision = off
  SafeModuleID = 52
  DigitalOutput01 = viaSafeLOGIC
  DigitalOutput02 = viaSafeLOGIC
  DigitalOutput03 = viaSafeLOGIC
  DigitalOutput04 = viaSafeLOGIC
X20SO4120_400_SC03 : X20SO4120 v2.2.1.0  [SS1 -> X20TB52d.SS; SL -> X20BM33b.SL1]
  Supervision = off
  SafeModuleID = 53
  DigitalOutput01 = viaSafeLOGIC
  DigitalOutput02 = viaSafeLOGIC
  DigitalOutput03 = viaSafeLOGIC
  DigitalOutput04 = viaSafeLOGIC
X20SO4120_400_SC04 : X20SO4120 v2.2.1.0  [SS1 -> X20TB52e.SS; SL -> X20BM33c.SL1]
  Supervision = off
  SafeModuleID = 54
  DigitalOutput01 = viaSafeLOGIC
  DigitalOutput02 = viaSafeLOGIC
  DigitalOutput03 = viaSafeLOGIC
  DigitalOutput04 = viaSafeLOGIC
X20SO4120_400_SC05 : X20SO4120 v2.2.1.0  [SS1 -> X20TB52f.SS; SL -> X20BM33e.SL1]
  Supervision = off
  SafeModuleID = 55
  DigitalOutput01 = viaSafeLOGIC
  DigitalOutput02 = viaSafeLOGIC
  DigitalOutput03 = viaSafeLOGIC
  DigitalOutput04 = viaSafeLOGIC
X20SO4120_MC01_K110 : X20SO4120 v2.2.1.0  [SS1 -> X20TB52a.SS; SL -> X20BM33.SL1]
  Supervision = off
  SafeModuleID = 3
  DigitalOutput01 = viaSafeLOGIC
  DigitalOutput02 = viaSafeLOGIC
  DigitalOutput03 = viaSafeLOGIC
  DigitalOutput04 = viaSafeLOGIC
X20SO4120_MC02_K109 : X20SO4120 v2.2.1.0  [SS1 -> X20TB52i.SS; SL -> X20BM33f.SL1]
  Supervision = off
  SafeModuleID = 5
  DigitalOutput01 = viaSafeLOGIC
  DigitalOutput02 = viaSafeLOGIC
  DigitalOutput03 = viaSafeLOGIC
  DigitalOutput04 = viaSafeLOGIC
X20SO4120_MC02_K110 : X20SO4120 v2.2.1.0  [SS1 -> X20TB52j.SS; SL -> X20BM33g.SL1]
  Supervision = off
  SafeModuleID = 6
  DigitalOutput01 = viaSafeLOGIC
  DigitalOutput02 = viaSafeLOGIC
  DigitalOutput03 = viaSafeLOGIC
  DigitalOutput04 = viaSafeLOGIC
X20SO4120_MC02_K111 : X20SO4120 v2.2.1.0  [SS1 -> X20TB52k.SS; SL -> X20BM33h.SL1]
  Supervision = off
  SafeModuleID = 8
  DigitalOutput01 = viaSafeLOGIC
  DigitalOutput02 = viaSafeLOGIC
  DigitalOutput03 = viaSafeLOGIC
  DigitalOutput04 = viaSafeLOGIC
X20TB12 : X20TB12 v1.0.0.0
X20TB12a : X20TB12 v1.0.0.0
X20TB12b : X20TB12 v1.0.0.0
X20TB12c : X20TB12 v1.0.0.0
X20TB12d : X20TB12 v1.0.0.0
X20TB12e : X20TB12 v1.0.0.0
X20TB12f : X20TB12 v1.0.0.0
X20TB12g : X20TB12 v1.0.0.0
X20TB12h : X20TB12 v1.0.0.0
X20TB12i : X20TB12 v1.0.0.0
X20TB12j : X20TB12 v1.0.0.0
X20TB12k : X20TB12 v1.0.0.0
X20TB12l : X20TB12 v1.0.0.0
X20TB12m : X20TB12 v1.0.0.0
X20TB12n : X20TB12 v1.0.0.0
X20TB12o : X20TB12 v1.0.0.0
X20TB12p : X20TB12 v1.0.0.0
X20TB12q : X20TB12 v1.0.0.0
X20TB12r : X20TB12 v1.0.0.0
X20TB12s : X20TB12 v1.0.0.0
X20TB12t : X20TB12 v1.0.0.0
X20TB52 : X20TB52 v1.0.0.2
X20TB52a : X20TB52 v1.0.0.2
X20TB52b : X20TB52 v1.0.0.2
X20TB52c : X20TB52 v1.0.0.2
X20TB52d : X20TB52 v1.0.0.2
X20TB52e : X20TB52 v1.0.0.2
X20TB52f : X20TB52 v1.0.0.2
X20TB52g : X20TB52 v1.0.0.2
X20TB52h : X20TB52 v1.0.0.2
X20TB52i : X20TB52 v1.0.0.2
X20TB52j : X20TB52 v1.0.0.2
X20TB52k : X20TB52 v1.0.0.2
X20ZF0000_MC01_K107 : X20ZF0000 v1.1.0.0  [SS1 -> X20TB12d.SS; SL -> X20BM11c.SL1]
X20ZF0000_MC01_K108 : X20ZF0000 v1.1.0.0  [SS1 -> X20TB12f.SS; SL -> X20BM11e.SL1]
X67AI2744_1801 : X67AI2744 v1.3.0.0  [X2X1 -> X67DM1321_1351.X2X2 [Cable Type=X2XCable, Length=10, Version=1.0.0.3]]
  Supervision = off
X67AI2744_1802 : X67AI2744 v1.3.0.0  [X2X1 -> X67DM1321_1354.X2X2 [Cable Type=X2XCable, Length=10, Version=1.0.0.3]]
  Supervision = off
X67AI2744_1803 : X67AI2744 v1.3.0.0  [X2X1 -> X67DM1321_1357.X2X2 [Cable Type=X2XCable, Length=10, Version=1.0.0.3]]
  Supervision = off
X67AI2744_1804 : X67AI2744 v1.3.0.0  [X2X1 -> X67DM1321_1360.X2X2 [Cable Type=X2XCable, Length=10, Version=1.0.0.3]]
  Supervision = off
X67AI2744_1805 : X67AI2744 v1.3.0.0  [X2X1 -> X67DM1321_1363.X2X2 [Cable Type=X2XCable, Length=10, Version=1.0.0.3]]
  Supervision = off
X67AI2744_1806 : X67AI2744 v1.3.0.0  [X2X1 -> X67DM1321_1366.X2X2 [Cable Type=X2XCable, Length=10, Version=1.0.0.3]]
  Supervision = off
X67AI2744_1807 : X67AI2744 v1.3.0.0  [X2X1 -> X67DM1321_1369.X2X2 [Cable Type=X2XCable, Length=10, Version=1.0.0.3]]
  Supervision = off
X67AI2744_1808 : X67AI2744 v1.3.0.0  [X2X1 -> X67DM1321_1372.X2X2 [Cable Type=X2XCable, Length=10, Version=1.0.0.3]]
  Supervision = off
X67AI2744_1809 : X67AI2744 v1.3.0.0  [X2X1 -> X67DM1321_1375.X2X2 [Cable Type=X2XCable, Length=10, Version=1.0.0.3]]
  Supervision = off
X67AI2744_1810 : X67AI2744 v1.3.0.0  [X2X1 -> X67DM1321_1378.X2X2 [Cable Type=X2XCable, Length=10, Version=1.0.0.3]]
  Supervision = off
X67AI2744_1811 : X67AI2744 v1.3.0.0  [X2X1 -> X67DM1321_1381.X2X2 [Cable Type=X2XCable, Length=10, Version=1.0.0.3]]
  Supervision = off
X67AI2744_1812 : X67AI2744 v1.3.0.0  [X2X1 -> X67DM1321_1384.X2X2 [Cable Type=X2XCable, Length=10, Version=1.0.0.3]]
  Supervision = off
X67AI2744_1813 : X67AI2744 v1.3.0.0  [X2X1 -> X67DM1321_1387.X2X2 [Cable Type=X2XCable, Length=10, Version=1.0.0.3]]
  Supervision = off
X67AI2744_1814 : X67AI2744 v1.3.0.0  [X2X1 -> X67DM1321_1390.X2X2 [Cable Type=X2XCable, Length=10, Version=1.0.0.3]]
  Supervision = off
X67AI2744_1815 : X67AI2744 v1.3.0.0  [X2X1 -> X67DM1321_1393.X2X2 [Cable Type=X2XCable, Length=10, Version=1.0.0.3]]
  Supervision = off
X67AI2744_1816 : X67AI2744 v1.3.0.0  [X2X1 -> X67DM1321_1396.X2X2 [Cable Type=X2XCable, Length=10, Version=1.0.0.3]]
  Supervision = off
X67AI2744_1817 : X67AI2744 v1.3.0.0  [X2X1 -> X67DM1321_1399.X2X2 [Cable Type=X2XCable, Length=10, Version=1.0.0.3]]
  Supervision = off
X67AI2744_1818 : X67AI2744 v1.3.0.0  [X2X1 -> X67DM1321_1602.X2X2 [Cable Type=X2XCable, Length=10, Version=1.0.0.3]]
  Supervision = off
X67AI2744_1819 : X67AI2744 v1.3.0.0  [X2X1 -> X67DM1321_1605.X2X2 [Cable Type=X2XCable, Length=10, Version=1.0.0.3]]
  Supervision = off
X67AI2744_1820 : X67AI2744 v1.3.0.0  [X2X1 -> X67DM1321_1608.X2X2 [Cable Type=X2XCable, Length=10, Version=1.0.0.3]]
  Supervision = off
X67AI2744_1821 : X67AI2744 v1.3.0.0  [X2X1 -> X67DM1321_1611.X2X2 [Cable Type=X2XCable, Length=10, Version=1.0.0.3]]
  Supervision = off
X67AI2744_1822 : X67AI2744 v1.3.0.0  [X2X1 -> X67DM1321_1614.X2X2 [Cable Type=X2XCable, Length=10, Version=1.0.0.3]]
  Supervision = off
X67AI2744_1823 : X67AI2744 v1.3.0.0  [X2X1 -> X67DM1321_1617.X2X2 [Cable Type=X2XCable, Length=10, Version=1.0.0.3]]
  Supervision = off
X67AI2744_1824 : X67AI2744 v1.3.0.0  [X2X1 -> X67DM1321_1620.X2X2 [Cable Type=X2XCable, Length=10, Version=1.0.0.3]]
  Supervision = off
X67AI2744_1825 : X67AI2744 v1.3.0.0  [X2X1 -> X67DM1321_1303.X2X2 [Cable Type=X2XCable, Length=10, Version=1.0.0.3]]
  Supervision = off
X67AI2744_1826 : X67AI2744 v1.3.0.0  [X2X1 -> X67DM1321_1304.X2X2 [Cable Type=X2XCable, Length=10, Version=1.0.0.3]]
  Supervision = off
X67AI2744_1827 : X67AI2744 v1.3.0.0  [X2X1 -> X67DM1321_1327.X2X2 [Cable Type=X2XCable, Length=10, Version=1.0.0.3]]
  Supervision = off
X67AI2744_1828 : X67AI2744 v1.3.0.0  [X2X1 -> X67DM1321_1328.X2X2 [Cable Type=X2XCable, Length=10, Version=1.0.0.3]]
  Supervision = off
X67AI2744_1829 : X67AI2744 v1.3.0.0  [X2X1 -> X67DM1321_1307.X2X2 [Cable Type=X2XCable, Length=10, Version=1.0.0.3]]
  Supervision = off
X67AI2744_1830 : X67AI2744 v1.3.0.0  [X2X1 -> X67DM1321_1308.X2X2 [Cable Type=X2XCable, Length=10, Version=1.0.0.3]]
  Supervision = off
X67AI2744_1831 : X67AI2744 v1.3.0.0  [X2X1 -> X67DM1321_1331.X2X2 [Cable Type=X2XCable, Length=10, Version=1.0.0.3]]
  Supervision = off
X67AI2744_1832 : X67AI2744 v1.3.0.0  [X2X1 -> X67DM1321_1332.X2X2 [Cable Type=X2XCable, Length=10, Version=1.0.0.3]]
  Supervision = off
X67AI2744_1833 : X67AI2744 v1.3.0.0  [X2X1 -> X67DM1321_1311.X2X2 [Cable Type=X2XCable, Length=10, Version=1.0.0.3]]
  Supervision = off
X67AI2744_1834 : X67AI2744 v1.3.0.0  [X2X1 -> X67DM1321_1312.X2X2 [Cable Type=X2XCable, Length=10, Version=1.0.0.3]]
  Supervision = off
X67AI2744_1835 : X67AI2744 v1.3.0.0  [X2X1 -> X67DM1321_1335.X2X2 [Cable Type=X2XCable, Length=10, Version=1.0.0.3]]
  Supervision = off
X67AI2744_1837 : X67AI2744 v1.3.0.0  [X2X1 -> X67DM1321_1315.X2X2 [Cable Type=X2XCable, Length=10, Version=1.0.0.3]]
  Supervision = off
X67AI2744_1838 : X67AI2744 v1.3.0.0  [X2X1 -> X67DM1321_1316.X2X2 [Cable Type=X2XCable, Length=10, Version=1.0.0.3]]
  Supervision = off
X67AI2744_1839 : X67AI2744 v1.3.0.0  [X2X1 -> X67DM1321_1339.X2X2 [Cable Type=X2XCable, Length=10, Version=1.0.0.3]]
  Supervision = off
X67AI2744_1841 : X67AI2744 v1.3.0.0  [X2X1 -> X67DM1321_1319.X2X2 [Cable Type=X2XCable, Length=10, Version=1.0.0.3]]
  Supervision = off
X67AI2744_1842 : X67AI2744 v1.3.0.0  [X2X1 -> X67DM1321_1320.X2X2 [Cable Type=X2XCable, Length=10, Version=1.0.0.3]]
  Supervision = off
X67AI2744_1843 : X67AI2744 v1.3.0.0  [X2X1 -> X67DM1321_1343.X2X2 [Cable Type=X2XCable, Length=10, Version=1.0.0.3]]
  Supervision = off
X67AI2744_1845 : X67AI2744 v1.3.0.0  [X2X1 -> X67DM1321_1323.X2X2 [Cable Type=X2XCable, Length=10, Version=1.0.0.3]]
  Supervision = off
X67AI2744_1846 : X67AI2744 v1.3.0.0  [X2X1 -> X67DM1321_1324.X2X2 [Cable Type=X2XCable, Length=10, Version=1.0.0.3]]
  Supervision = off
X67AI2744_1847 : X67AI2744 v1.3.0.0  [X2X1 -> X67DM1321_1347.X2X2 [Cable Type=X2XCable, Length=10, Version=1.0.0.3]]
  Supervision = off
X67BC8321_PL31 : X67BC8321-1 v2.11.1.0  [PLK1 -> 0AC808.9a.ETH4 (NodeNumber=31) [Cable Type=PowerlinkCable, Length=10, Version=1.0.0.3]]
  IOSupervision = off
X67BC8321_PL32 : X67BC8321-1 v2.11.1.0  [PLK1 -> 0AC808.9a.ETH1 (NodeNumber=32) [Cable Type=PowerlinkCable, Length=10, Version=1.0.0.3]]
  IOSupervision = off
X67BC8321_PL33 : X67BC8321-1 v2.11.1.0  [PLK1 -> 0AC808.9a.ETH2 (NodeNumber=33) [Cable Type=PowerlinkCable, Length=10, Version=1.0.0.3]]
  IOSupervision = off
X67BC8321_PL34 : X67BC8321-1 v2.11.1.0  [PLK1 -> 0AC808.9a.ETH3 (NodeNumber=34) [Cable Type=PowerlinkCable, Length=10, Version=1.0.0.3]]
  IOSupervision = off
X67BC8321_PL35 : X67BC8321-1 v2.11.1.0  [PLK1 -> 0AC808.9a.ETH5 (NodeNumber=35) [Cable Type=PowerlinkCable, Length=10, Version=1.0.0.3]]
  IOSupervision = off
X67BC8321_PL36 : X67BC8321-1 v2.11.1.0  [PLK1 -> 0AC808.9a.ETH6 (NodeNumber=36) [Cable Type=PowerlinkCable, Length=10, Version=1.0.0.3]]
  IOSupervision = off
X67BC8321_PL37 : X67BC8321-1 v2.11.1.0  [PLK1 -> 0AC808.9a.ETH7 (NodeNumber=37) [Cable Type=PowerlinkCable, Length=10, Version=1.0.0.3]]
  IOSupervision = off
X67BC8321_PL38 : X67BC8321-1 v2.11.1.0  [PLK1 -> 0AC808.9c.ETH1 (NodeNumber=38) [Cable Type=PowerlinkCable, Length=10, Version=1.0.0.3]]
  IOSupervision = off
X67BC8321_PL39 : X67BC8321-1 v2.11.1.0  [PLK1 -> 0AC808.9c.ETH2 (NodeNumber=39) [Cable Type=PowerlinkCable, Length=10, Version=1.0.0.3]]
  IOSupervision = off
X67BC8321_PL43_S : X67BC8321-1 v2.11.1.0  [PLK1 -> 0AC808.9c.ETH3 (NodeNumber=43) [Cable Type=PowerlinkCable, Length=10, Version=1.0.0.3]]
  IOSupervision = off
X67BC8321_PL44 : X67BC8321-1 v2.11.1.0  [PLK1 -> 0AC808.9c.ETH4 (NodeNumber=44) [Cable Type=PowerlinkCable, Length=10, Version=1.0.0.3]]
  IOSupervision = off
X67DM1321_1301 : X67DM1321 v1.2.0.0  [X2X1 -> X67BC8321_PL35.IF1 [Cable Type=X2XCable, Length=10, Version=1.0.0.3]]
  Supervision = off
  Direction04 = output
  Direction05 = output
  Direction06 = output
  Direction07 = output
X67DM1321_1302 : X67DM1321 v1.2.0.0  [X2X1 -> X67AI2744_1825.X2X2 [Cable Type=X2XCable, Length=10, Version=1.0.0.3]]
  Supervision = off
  Direction04 = output
  Direction05 = output
  Direction06 = output
  Direction07 = output
X67DM1321_1303 : X67DM1321 v1.2.0.0  [X2X1 -> X67DM1321_1301.X2X2 [Cable Type=X2XCable, Length=10, Version=1.0.0.3]]
  Supervision = off
  Direction04 = output
  Direction05 = output
  Direction06 = output
  Direction07 = output
X67DM1321_1304 : X67DM1321 v1.2.0.0  [X2X1 -> X67DM1321_1302.X2X2 [Cable Type=X2XCable, Length=10, Version=1.0.0.3]]
  Supervision = off
  Direction04 = output
  Direction05 = output
  Direction06 = output
  Direction07 = output
X67DM1321_1305 : X67DM1321 v1.2.0.0  [X2X1 -> X67AI2744_1828.X2X2 [Cable Type=X2XCable, Length=10, Version=1.0.0.3]]
  Supervision = off
  Direction04 = output
  Direction05 = output
  Direction06 = output
  Direction07 = output
X67DM1321_1306 : X67DM1321 v1.2.0.0  [X2X1 -> X67AI2744_1829.X2X2 [Cable Type=X2XCable, Length=10, Version=1.0.0.3]]
  Supervision = off
  Direction04 = output
  Direction05 = output
  Direction06 = output
  Direction07 = output
X67DM1321_1307 : X67DM1321 v1.2.0.0  [X2X1 -> X67DM1321_1305.X2X2 [Cable Type=X2XCable, Length=10, Version=1.0.0.3]]
  Supervision = off
  Direction04 = output
  Direction05 = output
  Direction06 = output
  Direction07 = output
X67DM1321_1308 : X67DM1321 v1.2.0.0  [X2X1 -> X67DM1321_1306.X2X2 [Cable Type=X2XCable, Length=10, Version=1.0.0.3]]
  Supervision = off
  Direction04 = output
  Direction05 = output
  Direction06 = output
  Direction07 = output
X67DM1321_1309 : X67DM1321 v1.2.0.0  [X2X1 -> X67BC8321_PL36.IF1 [Cable Type=X2XCable, Length=10, Version=1.0.0.3]]
  Supervision = off
  Direction04 = output
  Direction05 = output
  Direction06 = output
  Direction07 = output
X67DM1321_1310 : X67DM1321 v1.2.0.0  [X2X1 -> X67AI2744_1833.X2X2 [Cable Type=X2XCable, Length=10, Version=1.0.0.3]]
  Supervision = off
  Direction04 = output
  Direction05 = output
  Direction06 = output
  Direction07 = output
X67DM1321_1311 : X67DM1321 v1.2.0.0  [X2X1 -> X67DM1321_1309.X2X2 [Cable Type=X2XCable, Length=10, Version=1.0.0.3]]
  Supervision = off
  Direction04 = output
  Direction05 = output
  Direction06 = output
  Direction07 = output
X67DM1321_1312 : X67DM1321 v1.2.0.0  [X2X1 -> X67DM1321_1310.X2X2 [Cable Type=X2XCable, Length=10, Version=1.0.0.3]]
  Supervision = off
  Direction04 = output
  Direction05 = output
  Direction06 = output
  Direction07 = output
X67DM1321_1313 : X67DM1321 v1.2.0.0  [X2X1 -> X67BC8321_PL37.IF1 [Cable Type=X2XCable, Length=10, Version=1.0.0.3]]
  Supervision = off
  Direction04 = output
  Direction05 = output
  Direction06 = output
  Direction07 = output
X67DM1321_1314 : X67DM1321 v1.2.0.0  [X2X1 -> X67AI2744_1837.X2X2 [Cable Type=X2XCable, Length=10, Version=1.0.0.3]]
  Supervision = off
  Direction04 = output
  Direction05 = output
  Direction06 = output
  Direction07 = output
X67DM1321_1315 : X67DM1321 v1.2.0.0  [X2X1 -> X67DM1321_1313.X2X2 [Cable Type=X2XCable, Length=10, Version=1.0.0.3]]
  Supervision = off
  Direction04 = output
  Direction05 = output
  Direction06 = output
  Direction07 = output
X67DM1321_1316 : X67DM1321 v1.2.0.0  [X2X1 -> X67DM1321_1314.X2X2 [Cable Type=X2XCable, Length=10, Version=1.0.0.3]]
  Supervision = off
  Direction04 = output
  Direction05 = output
  Direction06 = output
  Direction07 = output
X67DM1321_1317 : X67DM1321 v1.2.0.0  [X2X1 -> X67DM1321_1340.X2X2 [Cable Type=X2XCable, Length=10, Version=1.0.0.3]]
  Supervision = off
  Direction04 = output
  Direction05 = output
  Direction06 = output
  Direction07 = output
X67DM1321_1318 : X67DM1321 v1.2.0.0  [X2X1 -> X67AI2744_1841.X2X2 [Cable Type=X2XCable, Length=10, Version=1.0.0.3]]
  Supervision = off
  Direction04 = output
  Direction05 = output
  Direction06 = output
  Direction07 = output
X67DM1321_1319 : X67DM1321 v1.2.0.0  [X2X1 -> X67DM1321_1317.X2X2 [Cable Type=X2XCable, Length=10, Version=1.0.0.3]]
  Supervision = off
  Direction04 = output
  Direction05 = output
  Direction06 = output
  Direction07 = output
X67DM1321_1320 : X67DM1321 v1.2.0.0  [X2X1 -> X67DM1321_1318.X2X2 [Cable Type=X2XCable, Length=10, Version=1.0.0.3]]
  Supervision = off
  Direction04 = output
  Direction05 = output
  Direction06 = output
  Direction07 = output
X67DM1321_1321 : X67DM1321 v1.2.0.0  [X2X1 -> X67BC8321_PL38.IF1 [Cable Type=X2XCable, Length=10, Version=1.0.0.3]]
  Supervision = off
  Direction04 = output
  Direction05 = output
  Direction06 = output
  Direction07 = output
X67DM1321_1322 : X67DM1321 v1.2.0.0  [X2X1 -> X67AI2744_1845.X2X2 [Cable Type=X2XCable, Length=10, Version=1.0.0.3]]
  Supervision = off
  Direction04 = output
  Direction05 = output
  Direction06 = output
  Direction07 = output
X67DM1321_1323 : X67DM1321 v1.2.0.0  [X2X1 -> X67DM1321_1321.X2X2 [Cable Type=X2XCable, Length=10, Version=1.0.0.3]]
  Supervision = off
  Direction04 = output
  Direction05 = output
  Direction06 = output
  Direction07 = output
X67DM1321_1324 : X67DM1321 v1.2.0.0  [X2X1 -> X67DM1321_1322.X2X2 [Cable Type=X2XCable, Length=10, Version=1.0.0.3]]
  Supervision = off
  Direction04 = output
  Direction05 = output
  Direction06 = output
  Direction07 = output
X67DM1321_1325 : X67DM1321 v1.2.0.0  [X2X1 -> X67AI2744_1826.X2X2 [Cable Type=X2XCable, Length=10, Version=1.0.0.3]]
  Supervision = off
  Direction04 = output
  Direction05 = output
  Direction06 = output
  Direction07 = output
X67DM1321_1326 : X67DM1321 v1.2.0.0  [X2X1 -> X67AI2744_1827.X2X2 [Cable Type=X2XCable, Length=10, Version=1.0.0.3]]
  Supervision = off
  Direction04 = output
  Direction05 = output
  Direction06 = output
  Direction07 = output
X67DM1321_1327 : X67DM1321 v1.2.0.0  [X2X1 -> X67DM1321_1325.X2X2 [Cable Type=X2XCable, Length=10, Version=1.0.0.3]]
  Supervision = off
  Direction04 = output
  Direction05 = output
  Direction06 = output
  Direction07 = output
X67DM1321_1328 : X67DM1321 v1.2.0.0  [X2X1 -> X67DM1321_1326.X2X2 [Cable Type=X2XCable, Length=10, Version=1.0.0.3]]
  Supervision = off
  Direction04 = output
  Direction05 = output
  Direction06 = output
  Direction07 = output
X67DM1321_1329 : X67DM1321 v1.2.0.0  [X2X1 -> X67AI2744_1830.X2X2 [Cable Type=X2XCable, Length=10, Version=1.0.0.3]]
  Supervision = off
  Direction04 = output
  Direction05 = output
  Direction06 = output
  Direction07 = output
X67DM1321_1330 : X67DM1321 v1.2.0.0  [X2X1 -> X67AI2744_1831.X2X2 [Cable Type=X2XCable, Length=10, Version=1.0.0.3]]
  Supervision = off
  Direction04 = output
  Direction05 = output
  Direction06 = output
  Direction07 = output
X67DM1321_1331 : X67DM1321 v1.2.0.0  [X2X1 -> X67DM1321_1329.X2X2 [Cable Type=X2XCable, Length=10, Version=1.0.0.3]]
  Supervision = off
  Direction04 = output
  Direction05 = output
  Direction06 = output
  Direction07 = output
X67DM1321_1332 : X67DM1321 v1.2.0.0  [X2X1 -> X67DM1321_1330.X2X2 [Cable Type=X2XCable, Length=10, Version=1.0.0.3]]
  Supervision = off
  Direction04 = output
  Direction05 = output
  Direction06 = output
  Direction07 = output
X67DM1321_1333 : X67DM1321 v1.2.0.0  [X2X1 -> X67AI2744_1834.X2X2 [Cable Type=X2XCable, Length=10, Version=1.0.0.3]]
  Supervision = off
  Direction04 = output
  Direction05 = output
  Direction06 = output
  Direction07 = output
X67DM1321_1334 : X67DM1321 v1.2.0.0  [X2X1 -> X67AI2744_1835.X2X2 [Cable Type=X2XCable, Length=10, Version=1.0.0.3]]
  Supervision = off
  Direction04 = output
  Direction05 = output
  Direction06 = output
  Direction07 = output
X67DM1321_1335 : X67DM1321 v1.2.0.0  [X2X1 -> X67DM1321_1333.X2X2 [Cable Type=X2XCable, Length=10, Version=1.0.0.3]]
  Supervision = off
  Direction04 = output
  Direction05 = output
  Direction06 = output
  Direction07 = output
X67DM1321_1336 : X67DM1321 v1.2.0.0  [X2X1 -> X67DM1321_1334.X2X2 [Cable Type=X2XCable, Length=10, Version=1.0.0.3]]
  Supervision = off
  Direction04 = output
  Direction05 = output
  Direction06 = output
  Direction07 = output
X67DM1321_1337 : X67DM1321 v1.2.0.0  [X2X1 -> X67AI2744_1838.X2X2 [Cable Type=X2XCable, Length=10, Version=1.0.0.3]]
  Supervision = off
  Direction04 = output
  Direction05 = output
  Direction06 = output
  Direction07 = output
X67DM1321_1338 : X67DM1321 v1.2.0.0  [X2X1 -> X67AI2744_1839.X2X2 [Cable Type=X2XCable, Length=10, Version=1.0.0.3]]
  Supervision = off
  Direction04 = output
  Direction05 = output
  Direction06 = output
  Direction07 = output
X67DM1321_1339 : X67DM1321 v1.2.0.0  [X2X1 -> X67DM1321_1337.X2X2 [Cable Type=X2XCable, Length=10, Version=1.0.0.3]]
  Supervision = off
  Direction04 = output
  Direction05 = output
  Direction06 = output
  Direction07 = output
X67DM1321_1340 : X67DM1321 v1.2.0.0  [X2X1 -> X67DM1321_1338.X2X2 [Cable Type=X2XCable, Length=10, Version=1.0.0.3]]
  Supervision = off
  Direction04 = output
  Direction05 = output
  Direction06 = output
  Direction07 = output
X67DM1321_1341 : X67DM1321 v1.2.0.0  [X2X1 -> X67AI2744_1842.X2X2 [Cable Type=X2XCable, Length=10, Version=1.0.0.3]]
  Supervision = off
  Direction04 = output
  Direction05 = output
  Direction06 = output
  Direction07 = output
X67DM1321_1342 : X67DM1321 v1.2.0.0  [X2X1 -> X67AI2744_1843.X2X2 [Cable Type=X2XCable, Length=10, Version=1.0.0.3]]
  Supervision = off
  Direction04 = output
  Direction05 = output
  Direction06 = output
  Direction07 = output
X67DM1321_1343 : X67DM1321 v1.2.0.0  [X2X1 -> X67DM1321_1341.X2X2 [Cable Type=X2XCable, Length=10, Version=1.0.0.3]]
  Supervision = off
  Direction04 = output
  Direction05 = output
  Direction06 = output
  Direction07 = output
X67DM1321_1344 : X67DM1321 v1.2.0.0  [X2X1 -> X67DM1321_1342.X2X2 [Cable Type=X2XCable, Length=10, Version=1.0.0.3]]
  Supervision = off
  Direction04 = output
  Direction05 = output
  Direction06 = output
  Direction07 = output
X67DM1321_1345 : X67DM1321 v1.2.0.0  [X2X1 -> X67AI2744_1846.X2X2 [Cable Type=X2XCable, Length=10, Version=1.0.0.3]]
  Supervision = off
  Direction04 = output
  Direction05 = output
  Direction06 = output
  Direction07 = output
X67DM1321_1346 : X67DM1321 v1.2.0.0  [X2X1 -> X67AI2744_1847.X2X2 [Cable Type=X2XCable, Length=10, Version=1.0.0.3]]
  Supervision = off
  Direction04 = output
  Direction05 = output
  Direction06 = output
  Direction07 = output
X67DM1321_1347 : X67DM1321 v1.2.0.0  [X2X1 -> X67DM1321_1345.X2X2 [Cable Type=X2XCable, Length=10, Version=1.0.0.3]]
  Supervision = off
  Direction04 = output
  Direction05 = output
  Direction06 = output
  Direction07 = output
X67DM1321_1348 : X67DM1321 v1.2.0.0  [X2X1 -> X67DM1321_1346.X2X2 [Cable Type=X2XCable, Length=10, Version=1.0.0.3]]
  Supervision = off
  Direction04 = output
  Direction05 = output
  Direction06 = output
  Direction07 = output
X67DM1321_1349 : X67DM1321 v1.2.0.0  [X2X1 -> X67BC8321_PL31.IF1 [Cable Type=X2XCable, Length=10, Version=1.0.0.3]]
  Supervision = off
  Direction05 = output
  Direction06 = output
  Direction07 = output
  Direction08 = output
X67DM1321_1351 : X67DM1321 v1.2.0.0  [X2X1 -> X67DM1321_1349.X2X2 [Cable Type=X2XCable, Length=10, Version=1.0.0.3]]
  Supervision = off
X67DM1321_1352 : X67DM1321 v1.2.0.0  [X2X1 -> X67AI2744_1801.X2X2 [Cable Type=X2XCable, Length=10, Version=1.0.0.3]]
  Supervision = off
  Direction05 = output
X67DM1321_1354 : X67DM1321 v1.2.0.0  [X2X1 -> X67DM1321_1352.X2X2 [Cable Type=X2XCable, Length=10, Version=1.0.0.3]]
  Supervision = off
X67DM1321_1355 : X67DM1321 v1.2.0.0  [X2X1 -> X67AI2744_1802.X2X2 [Cable Type=X2XCable, Length=10, Version=1.0.0.3]]
  Supervision = off
X67DM1321_1357 : X67DM1321 v1.2.0.0  [X2X1 -> X67DM1321_1355.X2X2 [Cable Type=X2XCable, Length=10, Version=1.0.0.3]]
  Supervision = off
X67DM1321_1358 : X67DM1321 v1.2.0.0  [X2X1 -> X67AI2744_1803.X2X2 [Cable Type=X2XCable, Length=10, Version=1.0.0.3]]
  Supervision = off
  Direction05 = output
  Direction06 = output
  Direction07 = output
  Direction08 = output
X67DM1321_1360 : X67DM1321 v1.2.0.0  [X2X1 -> X67DM1321_1358.X2X2 [Cable Type=X2XCable, Length=10, Version=1.0.0.3]]
  Supervision = off
X67DM1321_1361 : X67DM1321 v1.2.0.0  [X2X1 -> X67AI2744_1804.X2X2 [Cable Type=X2XCable, Length=10, Version=1.0.0.3]]
  Supervision = off
  Direction05 = output
X67DM1321_1363 : X67DM1321 v1.2.0.0  [X2X1 -> X67DM1321_1361.X2X2 [Cable Type=X2XCable, Length=10, Version=1.0.0.3]]
  Supervision = off
X67DM1321_1364 : X67DM1321 v1.2.0.0  [X2X1 -> X67AI2744_1805.X2X2 [Cable Type=X2XCable, Length=10, Version=1.0.0.3]]
  Supervision = off
X67DM1321_1366 : X67DM1321 v1.2.0.0  [X2X1 -> X67DM1321_1364.X2X2 [Cable Type=X2XCable, Length=10, Version=1.0.0.3]]
  Supervision = off
X67DM1321_1367 : X67DM1321 v1.2.0.0  [X2X1 -> X67BC8321_PL32.IF1 [Cable Type=X2XCable, Length=10, Version=1.0.0.3]]
  Supervision = off
  Direction05 = output
  Direction06 = output
  Direction07 = output
  Direction08 = output
X67DM1321_1369 : X67DM1321 v1.2.0.0  [X2X1 -> X67DM1321_1367.X2X2 [Cable Type=X2XCable, Length=10, Version=1.0.0.3]]
  Supervision = off
X67DM1321_1370 : X67DM1321 v1.2.0.0  [X2X1 -> X67AI2744_1807.X2X2 [Cable Type=X2XCable, Length=10, Version=1.0.0.3]]
  Supervision = off
  Direction05 = output
X67DM1321_1372 : X67DM1321 v1.2.0.0  [X2X1 -> X67DM1321_1370.X2X2 [Cable Type=X2XCable, Length=10, Version=1.0.0.3]]
  Supervision = off
X67DM1321_1373 : X67DM1321 v1.2.0.0  [X2X1 -> X67AI2744_1808.X2X2 [Cable Type=X2XCable, Length=10, Version=1.0.0.3]]
  Supervision = off
X67DM1321_1375 : X67DM1321 v1.2.0.0  [X2X1 -> X67DM1321_1373.X2X2 [Cable Type=X2XCable, Length=10, Version=1.0.0.3]]
  Supervision = off
X67DM1321_1376 : X67DM1321 v1.2.0.0  [X2X1 -> X67AI2744_1809.X2X2 [Cable Type=X2XCable, Length=10, Version=1.0.0.3]]
  Supervision = off
  Direction05 = output
  Direction06 = output
  Direction07 = output
  Direction08 = output
X67DM1321_1378 : X67DM1321 v1.2.0.0  [X2X1 -> X67DM1321_1376.X2X2 [Cable Type=X2XCable, Length=10, Version=1.0.0.3]]
  Supervision = off
X67DM1321_1379 : X67DM1321 v1.2.0.0  [X2X1 -> X67AI2744_1810.X2X2 [Cable Type=X2XCable, Length=10, Version=1.0.0.3]]
  Supervision = off
  Direction05 = output
X67DM1321_1381 : X67DM1321 v1.2.0.0  [X2X1 -> X67DM1321_1379.X2X2 [Cable Type=X2XCable, Length=10, Version=1.0.0.3]]
  Supervision = off
X67DM1321_1382 : X67DM1321 v1.2.0.0  [X2X1 -> X67AI2744_1811.X2X2 [Cable Type=X2XCable, Length=10, Version=1.0.0.3]]
  Supervision = off
X67DM1321_1384 : X67DM1321 v1.2.0.0  [X2X1 -> X67DM1321_1382.X2X2 [Cable Type=X2XCable, Length=10, Version=1.0.0.3]]
  Supervision = off
X67DM1321_1385 : X67DM1321 v1.2.0.0  [X2X1 -> X67BC8321_PL33.IF1 [Cable Type=X2XCable, Length=10, Version=1.0.0.3]]
  Supervision = off
  Direction05 = output
  Direction06 = output
  Direction07 = output
  Direction08 = output
X67DM1321_1387 : X67DM1321 v1.2.0.0  [X2X1 -> X67DM1321_1385.X2X2 [Cable Type=X2XCable, Length=10, Version=1.0.0.3]]
  Supervision = off
X67DM1321_1388 : X67DM1321 v1.2.0.0  [X2X1 -> X67AI2744_1813.X2X2 [Cable Type=X2XCable, Length=10, Version=1.0.0.3]]
  Supervision = off
  Direction05 = output
X67DM1321_1390 : X67DM1321 v1.2.0.0  [X2X1 -> X67DM1321_1388.X2X2 [Cable Type=X2XCable, Length=10, Version=1.0.0.3]]
  Supervision = off
X67DM1321_1391 : X67DM1321 v1.2.0.0  [X2X1 -> X67AI2744_1814.X2X2 [Cable Type=X2XCable, Length=10, Version=1.0.0.3]]
  Supervision = off
X67DM1321_1393 : X67DM1321 v1.2.0.0  [X2X1 -> X67DM1321_1391.X2X2 [Cable Type=X2XCable, Length=10, Version=1.0.0.3]]
  Supervision = off
X67DM1321_1394 : X67DM1321 v1.2.0.0  [X2X1 -> X67AI2744_1815.X2X2 [Cable Type=X2XCable, Length=10, Version=1.0.0.3]]
  Supervision = off
  Direction05 = output
  Direction06 = output
  Direction07 = output
  Direction08 = output
X67DM1321_1396 : X67DM1321 v1.2.0.0  [X2X1 -> X67DM1321_1394.X2X2 [Cable Type=X2XCable, Length=10, Version=1.0.0.3]]
  Supervision = off
X67DM1321_1397 : X67DM1321 v1.2.0.0  [X2X1 -> X67AI2744_1816.X2X2 [Cable Type=X2XCable, Length=10, Version=1.0.0.3]]
  Supervision = off
  Direction05 = output
X67DM1321_1399 : X67DM1321 v1.2.0.0  [X2X1 -> X67DM1321_1397.X2X2 [Cable Type=X2XCable, Length=10, Version=1.0.0.3]]
  Supervision = off
X67DM1321_1501 : X67DM1321 v1.2.0.0  [X2X1 -> X67SI8103_1401.X2X2 [Cable Type=X2XCable, Length=10, Version=1.0.0.3]]
  Supervision = off
  Direction01 = output
  Direction02 = output
  Direction03 = output
  Direction04 = output
  Direction05 = output
  Direction06 = output
  Direction07 = output
  Direction08 = output
X67DM1321_1502 : X67DM1321 v1.2.0.0  [X2X1 -> X67SI8103_1402.X2X2 [Cable Type=X2XCable, Length=10, Version=1.0.0.3]]
  Supervision = off
  Direction01 = output
  Direction02 = output
  Direction03 = output
  Direction04 = output
  Direction05 = output
  Direction06 = output
  Direction07 = output
  Direction08 = output
X67DM1321_1504 : X67DM1321 v1.2.0.0  [X2X1 -> X67SI8103_1404.X2X2 [Cable Type=X2XCable, Length=10, Version=1.0.0.3]]
  Supervision = off
X67DM1321_1506 : X67DM1321 v1.2.0.0  [X2X1 -> X67SI8103_1406.X2X2 [Cable Type=X2XCable, Length=10, Version=1.0.0.3]]
  Supervision = off
X67DM1321_1508 : X67DM1321 v1.2.0.0  [X2X1 -> X67SI8103_1408.X2X2 [Cable Type=X2XCable, Length=10, Version=1.0.0.3]]
  Supervision = off
  Direction01 = output
  Direction02 = output
  Direction03 = output
  Direction04 = output
  Direction05 = output
  Direction06 = output
  Direction07 = output
  Direction08 = output
X67DM1321_1509 : X67DM1321 v1.2.0.0  [X2X1 -> X67SI8103_1409.X2X2 [Cable Type=X2XCable, Length=10, Version=1.0.0.3]]
  Supervision = off
X67DM1321_1510 : X67DM1321 v1.2.0.0  [X2X1 -> X67SI8103_1410.X2X2 [Cable Type=X2XCable, Length=10, Version=1.0.0.3]]
  Supervision = off
  Direction06 = output
  Direction07 = output
  Direction08 = output
X67DM1321_1511 : X67DM1321 v1.2.0.0  [X2X1 -> X67SI8103_1411.X2X2 [Cable Type=X2XCable, Length=10, Version=1.0.0.3]]
  Supervision = off
  Direction01 = output
  Direction02 = output
  Direction03 = output
  Direction04 = output
  Direction05 = output
  Direction06 = output
  Direction07 = output
  Direction08 = output
X67DM1321_1514 : X67DM1321 v1.2.0.0  [X2X1 -> X67SI8103_1414.X2X2 [Cable Type=X2XCable, Length=10, Version=1.0.0.3]]
  Supervision = off
X67DM1321_1515 : X67DM1321 v1.2.0.0  [X2X1 -> X67SI8103_1415.X2X2 [Cable Type=X2XCable, Length=10, Version=1.0.0.3]]
  Supervision = off
X67DM1321_1600 : X67DM1321 v1.2.0.0  [X2X1 -> X67AI2744_1817.X2X2 [Cable Type=X2XCable, Length=10, Version=1.0.0.3]]
  Supervision = off
X67DM1321_1602 : X67DM1321 v1.2.0.0  [X2X1 -> X67DM1321_1600.X2X2 [Cable Type=X2XCable, Length=10, Version=1.0.0.3]]
  Supervision = off
X67DM1321_1603 : X67DM1321 v1.2.0.0  [X2X1 -> X67BC8321_PL34.IF1 [Cable Type=X2XCable, Length=10, Version=1.0.0.3]]
  Supervision = off
  Direction05 = output
  Direction06 = output
  Direction07 = output
  Direction08 = output
X67DM1321_1605 : X67DM1321 v1.2.0.0  [X2X1 -> X67DM1321_1603.X2X2 [Cable Type=X2XCable, Length=10, Version=1.0.0.3]]
  Supervision = off
X67DM1321_1606 : X67DM1321 v1.2.0.0  [X2X1 -> X67AI2744_1819.X2X2 [Cable Type=X2XCable, Length=10, Version=1.0.0.3]]
  Supervision = off
  Direction05 = output
X67DM1321_1608 : X67DM1321 v1.2.0.0  [X2X1 -> X67DM1321_1606.X2X2 [Cable Type=X2XCable, Length=10, Version=1.0.0.3]]
  Supervision = off
X67DM1321_1609 : X67DM1321 v1.2.0.0  [X2X1 -> X67AI2744_1820.X2X2 [Cable Type=X2XCable, Length=10, Version=1.0.0.3]]
  Supervision = off
X67DM1321_1611 : X67DM1321 v1.2.0.0  [X2X1 -> X67DM1321_1609.X2X2 [Cable Type=X2XCable, Length=10, Version=1.0.0.3]]
  Supervision = off
X67DM1321_1612 : X67DM1321 v1.2.0.0  [X2X1 -> X67AI2744_1821.X2X2 [Cable Type=X2XCable, Length=10, Version=1.0.0.3]]
  Supervision = off
  Direction05 = output
  Direction06 = output
  Direction07 = output
  Direction08 = output
X67DM1321_1614 : X67DM1321 v1.2.0.0  [X2X1 -> X67DM1321_1612.X2X2 [Cable Type=X2XCable, Length=10, Version=1.0.0.3]]
  Supervision = off
X67DM1321_1615 : X67DM1321 v1.2.0.0  [X2X1 -> X67AI2744_1822.X2X2 [Cable Type=X2XCable, Length=10, Version=1.0.0.3]]
  Supervision = off
  Direction05 = output
X67DM1321_1617 : X67DM1321 v1.2.0.0  [X2X1 -> X67DM1321_1615.X2X2 [Cable Type=X2XCable, Length=10, Version=1.0.0.3]]
  Supervision = off
X67DM1321_1618 : X67DM1321 v1.2.0.0  [X2X1 -> X67AI2744_1823.X2X2 [Cable Type=X2XCable, Length=10, Version=1.0.0.3]]
  Supervision = off
X67DM1321_1620 : X67DM1321 v1.2.0.0  [X2X1 -> X67DM1321_1618.X2X2 [Cable Type=X2XCable, Length=10, Version=1.0.0.3]]
  Supervision = off
X67DM1321_1625 : X67DM1321 v1.2.0.0  [X2X1 -> X67BC8321_PL39.IF1 [Cable Type=X2XCable, Length=10, Version=1.0.0.3]]
  Supervision = off
  Direction04 = output
  Direction05 = output
  Direction06 = output
  Direction07 = output
X67DM1321_1626 : X67DM1321 v1.2.0.0  [X2X1 -> X67DM1321_1625.X2X2 [Cable Type=X2XCable, Length=10, Version=1.0.0.3]]
  Supervision = off
  Direction04 = output
  Direction05 = output
  Direction06 = output
  Direction07 = output
X67DM1321_1627 : X67DM1321 v1.2.0.0  [X2X1 -> X67DM1321_1626.X2X2 [Cable Type=X2XCable, Length=10, Version=1.0.0.3]]
  Supervision = off
  Direction04 = output
  Direction05 = output
  Direction06 = output
  Direction07 = output
X67DM1321_1628 : X67DM1321 v1.2.0.0  [X2X1 -> X67DM1321_1627.X2X2 [Cable Type=X2XCable, Length=10, Version=1.0.0.3]]
  Supervision = off
  Direction04 = output
  Direction05 = output
  Direction06 = output
  Direction07 = output
X67DM1321_1630 : X67DM1321 v1.2.0.0  [X2X1 -> X67DM1321_1628.X2X2 [Cable Type=X2XCable, Length=10, Version=1.0.0.3]]
  Supervision = off
  Direction04 = output
  Direction05 = output
  Direction06 = output
  Direction07 = output
X67DM1321_1631 : X67DM1321 v1.2.0.0  [X2X1 -> X67DM1321_1630.X2X2 [Cable Type=X2XCable, Length=10, Version=1.0.0.3]]
  Supervision = off
  Direction04 = output
  Direction05 = output
  Direction06 = output
  Direction07 = output
X67SI8103_1401 : X67SI8103 v2.3.1.0  [X2X1 -> X67DM1321_1502.X2X2 [Cable Type=X2XCable, Length=10, Version=1.0.0.3]]
  Supervision = off
  SafeModuleID = 31
X67SI8103_1402 : X67SI8103 v2.3.1.0  [X2X1 -> X67BC8321_PL44.IF1 [Cable Type=X2XCable, Length=10, Version=1.0.0.3]]
  Supervision = off
  SafeModuleID = 32
X67SI8103_1403 : X67SI8103 v2.3.1.0  [X2X1 -> X67DM1321_1501.X2X2 [Cable Type=X2XCable, Length=10, Version=1.0.0.3]]
  Supervision = off
  SafeModuleID = 33
X67SI8103_1404 : X67SI8103 v2.3.1.0  [X2X1 -> X67DM1321_1515.X2X2 [Cable Type=X2XCable, Length=10, Version=1.0.0.3]]
  Supervision = off
  SafeModuleID = 34
X67SI8103_1406 : X67SI8103 v2.3.1.0  [X2X1 -> X67DM1321_1504.X2X2 [Cable Type=X2XCable, Length=10, Version=1.0.0.3]]
  Supervision = off
  SafeModuleID = 36
X67SI8103_1408 : X67SI8103 v2.3.1.0  [X2X1 -> X67SI8103_1416.X2X2 [Cable Type=X2XCable, Length=10, Version=1.0.0.3]]
  Supervision = off
  SafeModuleID = 7
X67SI8103_1409 : X67SI8103 v2.3.1.0  [X2X1 -> X67DM1321_1511.X2X2 [Cable Type=X2XCable, Length=10, Version=1.0.0.3]]
  Supervision = off
  SafeModuleID = 39
X67SI8103_1410 : X67SI8103 v2.3.1.0  [X2X1 -> X67DM1321_1508.X2X2 [Cable Type=X2XCable, Length=10, Version=1.0.0.3]]
  Supervision = off
  SafeModuleID = 40
X67SI8103_1411 : X67SI8103 v2.3.1.0  [X2X1 -> X67SI8103_1403.X2X2 [Cable Type=X2XCable, Length=10, Version=1.0.0.3]]
  Supervision = off
  SafeModuleID = 41
X67SI8103_1414 : X67SI8103 v2.3.1.0  [X2X1 -> X67BC8321_PL43_S.IF1 [Cable Type=X2XCable, Length=10, Version=1.0.0.3]]
  Supervision = off
  SafeModuleID = 44
X67SI8103_1415 : X67SI8103 v2.3.1.0  [X2X1 -> X67DM1321_1514.X2X2 [Cable Type=X2XCable, Length=10, Version=1.0.0.3]]
  Supervision = off
  SafeModuleID = 45
X67SI8103_1416 : X67SI8103 v2.3.1.0  [X2X1 -> X67DM1321_1509.X2X2 [Cable Type=X2XCable, Length=10, Version=1.0.0.3]]
  Supervision = off
  SafeModuleID = 46
```

### Cpu.per - APC2200/Cpu.per
```iecst
(********************************************************************
 * COPYRIGHT --
 ********************************************************************
 * File: Cpu.per
 * Author: Dave
 * Created: November 19, 2010
 ********************************************************************
 * Declaration of permanent variables
 ********************************************************************)
VAR_CONFIG
	gSettings AT %M0; (* *)
END_VAR
```
